// -------------------------------------------------
// subphase timer & counter
      A     M    103.0;

// -------------------------------------------------
// subphase actuator
      A     M    103.3;

// -------------------------------------------------
// subphase transition
      CLR   ;
      =     M    103.1;
      JU    COMM;
NETWORK
TITLE =phase 32: CIP Push Out
//SFM   Use                                 Datatype        UoM
//----+-------------------------------------------------------------------------
// 00 : Watch Dog Time                      Duration        min
// 01 : Step Time                           Duration        min
// 06 : Delay Switchpoint                   Duration        s
// 15 : Amount                              Value           m3
// 26 : CIP Step On Condition               Enumeration     min
// 27 : CIP Prerun                          Enumeration     min
// 28 : CIP Return                          Enumeration     min
// 29 : CIP Pump Speed                      Value           %
// 30 : CIP Return Temperature              Value           °C
// 32 : CIP Return Conductivity             Value           mS
// 34 : CIP Prerun Flow                     Value           m3/h
// 35 : CIP Prerun Pressure                 Value           bar
// 37 : CIP Pump Mode                       Enumeration     min
X32:  SET   ;
// ---------------------------------------------------------------------------
// General CM evaluation
      CALL FC   150 (
           ChkType                  := 3,
           ChkOK                    := #ChkOK);

      AN    #ChkOK;
      S     M    120.3;

// ---------------------------------------------------------------------------
// index evaluation: CIP Step On Condition
      CALL FC    45 (
           SFM                      := #U.Seq.SFM[26].Sp,
           Indexes                  := #S2I.SFM26);

// ---------------------------------------------------------------------------
// index evaluation: CIP Prerun
      CALL FC    45 (
           SFM                      := #U.Seq.SFM[27].Sp,
           Indexes                  := #S2I.SFM27);

// ---------------------------------------------------------------------------
// index evaluation: CIP Return
      CALL FC    45 (
           SFM                      := #U.Seq.SFM[28].Sp,
           Indexes                  := #S2I.SFM28);

// ---------------------------------------------------------------------------
// index evaluation: CIP Pump Mode
      CALL FC    45 (
           SFM                      := #U.Seq.SFM[37].Sp,
           Indexes                  := #S2I.SFM37);

// ---------------------------------------------------------------------------
// general functions
      AN    M    121.2;
      A     M    102.3;
      =     #RRel;

// ---------------------------------------------------------------------------
// messages
// ---------------------------------------------------------------------------
// timer & counter
      A     M    102.0;

// ---------------------------------------------------------------------------
// pause timer
      ON    M    102.3;
      O     M    150.0;
      S     M    140.0; // Step Time

      ON    M    102.3;
      O     M    150.5;
      S     M    140.5; // Delay Switchpoint

// ---------------------------------------------------------------------------
// communication

// ---------------------------------------------------------------------------
// control modules
      A     M    102.3;

// ---------------------------------------------------------------------------
// transition condition
      A     #SubStepMaxD;
      =     M    102.1;

// subphase evaluation
      L     MW   110;
      JL    D200;
      JU    COMM; // subphase  0:
// ---------------------------------------------------------------------------
D200: SET   ;
      S     M    110.7; // Error unknown subphase
      JU    COMM;
NETWORK
TITLE =phase 34: CIP Rinsing
//SFM   Use                                 Datatype        UoM
//----+-------------------------------------------------------------------------
// 00 : Watch Dog Time                      Duration        min
// 01 : Step Time                           Duration        min
// 05 : Substep Time                        Duration        s
// 06 : Delay Switchpoint                   Duration        s
// 15 : Amount                              Value           m3
// 27 : CIP Prerun                          Enumeration     min
// 28 : CIP Return                          Enumeration     min
// 29 : CIP Pump Speed                      Value           %
// 30 : CIP Return Temperature              Value           °C
// 32 : CIP Return Conductivity             Value           mS
// 34 : CIP Prerun Flow                     Value           m3/h
// 35 : CIP Prerun Pressure                 Value           bar
// 37 : CIP Pump Mode                       Enumeration     min
// 59 : Interval Counter                    Value           No.
X34:  SET   ;
// ---------------------------------------------------------------------------
// General CM evaluation
      CALL FC   150 (
           ChkType                  := 3,
           ChkOK                    := #ChkOK);

      AN    #ChkOK;
      S     M    120.3;

// ---------------------------------------------------------------------------
// index evaluation: CIP Prerun
      CALL FC    45 (
           SFM                      := #U.Seq.SFM[27].Sp,
           Indexes                  := #S2I.SFM27);

// ---------------------------------------------------------------------------
// index evaluation: CIP Return
      CALL FC    45 (
           SFM                      := #U.Seq.SFM[28].Sp,
           Indexes                  := #S2I.SFM28);

// ---------------------------------------------------------------------------
// index evaluation: CIP Pump Mode
      CALL FC    45 (
           SFM                      := #U.Seq.SFM[37].Sp,
           Indexes                  := #S2I.SFM37);

// ---------------------------------------------------------------------------
// general functions
      AN    M    121.2;
      A     M    102.3;
      =     #RRel;

// ---------------------------------------------------------------------------
// messages
// ---------------------------------------------------------------------------
// timer & counter
      A     M    102.0;

// ---------------------------------------------------------------------------
// pause timer
      ON    M    102.3;
      O     M    150.0;
      S     M    140.0; // Step Time

      ON    M    102.3;
      O     M    150.4;
      S     M    140.4; // Substep Time

      ON    M    102.3;
      O     M    150.5;
      S     M    140.5; // Delay Switchpoint

// ---------------------------------------------------------------------------
// communication

// ---------------------------------------------------------------------------
// control modules
      A     M    102.3;

// ---------------------------------------------------------------------------
// transition condition
      A     #SubStepMaxD;
      =     M    102.1;

// ---------------------------------------------------------------------------
// ---------------------------------------------------------------------------
// subphase repeat function
//      A     #SubStepMax
//      JCN  Y34
//      L     1
//      T     "SOSubStepNew"
//Y34:  SET

// subphase evaluation
      L     MW   110;
      JL    D400;
      JU    COMM; // subphase  0:
      JU    D401; // subphase  1: Pause
      JU    D402; // subphase  2: Main
      JU    D403; // subphase  3: Expulse
      JU    D404; // subphase  4: Seat Lift
      JU    D400; // subphase  5:
      JU    D406; // subphase  6: Shaft Rinse
      JU    D407; // subphase  7: Drain
// ---------------------------------------------------------------------------
D400: SET   ;
      S     M    110.7; // Error unknown subphase
      JU    COMM;

// subphase 1: Pause
D401: SET   ;

// -------------------------------------------------
// subphase timer & counter
      A     M    103.0;

// -------------------------------------------------
// subphase actuator
      A     M    103.3;

// -------------------------------------------------
// subphase transition
      CLR   ;
      =     M    103.1;
      JU    COMM;

// subphase 2: Main
D402: SET   ;

// -------------------------------------------------
// subphase timer & counter
      A     M    103.0;

// -------------------------------------------------
// subphase actuator
      A     M    103.3;

// -------------------------------------------------
// subphase transition
      CLR   ;
      =     M    103.1;
      JU    COMM;

// subphase 3: Expulse
D403: SET   ;

// -------------------------------------------------
// subphase timer & counter
      A     M    103.0;

// -------------------------------------------------
// subphase actuator
      A     M    103.3;

// -------------------------------------------------
// subphase transition
      CLR   ;
      =     M    103.1;
      JU    COMM;

// subphase 4: Seat Lift
D404: SET   ;

// -------------------------------------------------
// subphase timer & counter
      A     M    103.0;

// -------------------------------------------------
// subphase actuator
      A     M    103.3;

// -------------------------------------------------
// subphase transition
      CLR   ;
      =     M    103.1;
      JU    COMM;

// subphase 6: Shaft Rinse
D406: SET   ;

// -------------------------------------------------
// subphase timer & counter
      A     M    103.0;

// -------------------------------------------------
// subphase actuator
      A     M    103.3;

// -------------------------------------------------
// subphase transition
      CLR   ;
      =     M    103.1;
      JU    COMM;

// subphase 7: Drain
D407: SET   ;

// -------------------------------------------------
// subphase timer & counter
      A     M    103.0;

// -------------------------------------------------
// subphase actuator
      A     M    103.3;

// -------------------------------------------------
// subphase transition
      CLR   ;
      =     M    103.1;
      JU    COMM;
NETWORK
TITLE =phase 36: CIP Drain
//SFM   Use                                 Datatype        UoM
//----+-------------------------------------------------------------------------
// 00 : Watch Dog Time                      Duration        Min
// 04 : Delay Empty                         Duration        #sec
X36:  SET   ;
// ---------------------------------------------------------------------------
// General CM evaluation
      CALL FC   150 (
           ChkType                  := 3,
           ChkOK                    := #ChkOK);

      AN    #ChkOK;
      S     M    120.3;

// ---------------------------------------------------------------------------
// general functions
      AN    M    121.2;
      A     M    102.3;
      =     #RRel;

// ---------------------------------------------------------------------------
// messages
// ---------------------------------------------------------------------------
// timer & counter
      A     M    102.0;

// ---------------------------------------------------------------------------
// pause timer
      ON    M    102.3;
      O     M    150.3;
      S     M    140.3; // Delay Empty

// ---------------------------------------------------------------------------
// communication

// ---------------------------------------------------------------------------
// control modules
      A     M    102.3;

// ---------------------------------------------------------------------------
// transition condition
      A     #SubStepMaxD;
      =     M    102.1;

// subphase evaluation
      L     MW   110;
      JL    D600;
      JU    COMM; // subphase  0:
// ---------------------------------------------------------------------------
D600: SET   ;
      S     M    110.7; // Error unknown subphase
      JU    COMM;
NETWORK
TITLE =phase 40: CIP End
//SFM   Use                                 Datatype        UoM
//----+-------------------------------------------------------------------------
// 00 : Watch Dog Time                      Duration        min
X40:  SET   ;
// ---------------------------------------------------------------------------
// General CM evaluation
      CALL FC   150 (
           ChkType                  := 3,
           ChkOK                    := #ChkOK);

      AN    #ChkOK;
      S     M    120.3;

// ---------------------------------------------------------------------------
// general functions
      AN    M    121.2;
      A     M    102.3;
      =     #RRel;

// ---------------------------------------------------------------------------
// messages
// ---------------------------------------------------------------------------
// timer & counter
      A     M    102.0;

// ---------------------------------------------------------------------------
// pause timer
// ---------------------------------------------------------------------------
// communication

// ---------------------------------------------------------------------------
// control modules
      A     M    102.3;

// ---------------------------------------------------------------------------
// transition condition
      A     #SubStepMaxD;
      =     M    102.1;

// subphase evaluation
      L     MW   110;
      JL    E000;
      JU    COMM; // subphase  0:
// ---------------------------------------------------------------------------
E000: SET   ;
      S     M    110.7; // Error unknown subphase
      JU    COMM;

NETWORK
TITLE =End Of Sequence Organisation

COMM: SET   ;

// ---------------------------------------------------------------------------
// pause timer unit parameter

// Request Mole Water
      O     DB250.DBX  182.6;
      S     DB155.DBX   27.2;

      AN    DB1595.DBX   26.4; // Molchwasser
      R     DB250.DBX  188.0;

// Quelle
      L     DB155.DBW  254;
      L     1000;
      *I    ;
      T     #iTmp;

      L     0;
      T     #U.Seq.SFM[14].Sp;
      L     DB155.DBW  256;
      <I    ;
      JCN   ntru;
      L     #iTmp;
      +I    ;
      ITD   ;
      DTR   ;
      T     #U.Seq.SFM[14].Sp;
ntru: NOP   0;


NETWORK
TITLE =General Post Phase Controls
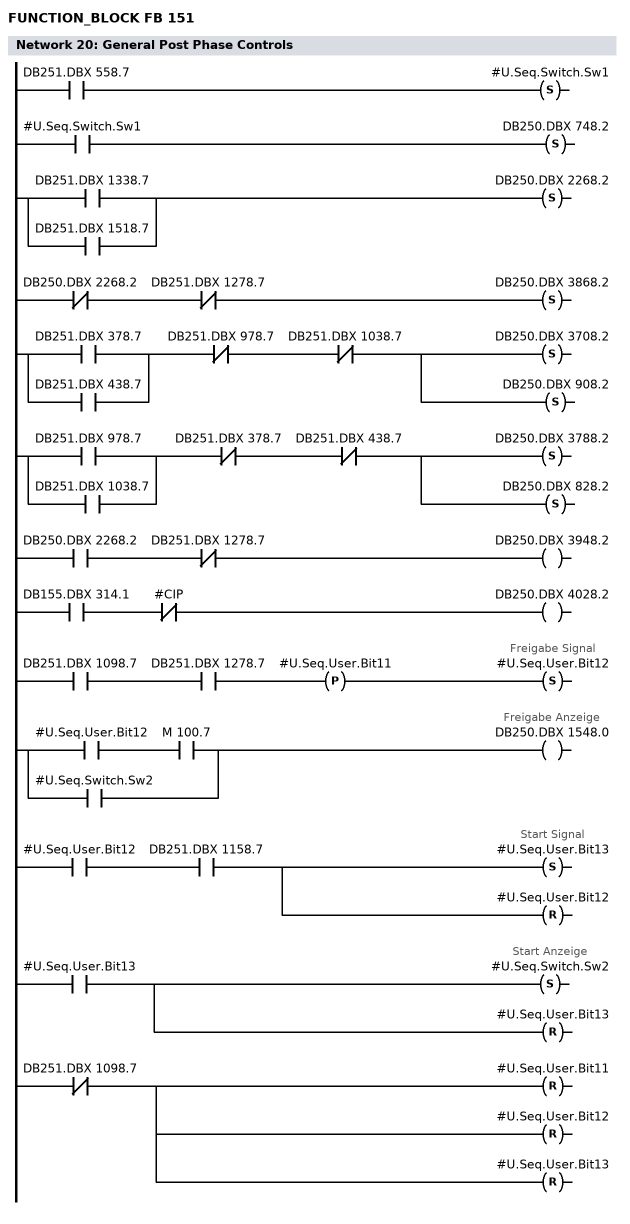

      NOP   0;

// ---------------------------------------------------------------------------
// general postphase controls
// Molchsignale  SR
      A     DB251.DBX  558.7;
      S     #U.Seq.Switch.Sw1;

      A     #U.Seq.Switch.Sw1;
      S     DB250.DBX  748.2;

// Molch Schwenkbogen auf CIP
      A     DB251.DBX 1338.7;
      O     DB251.DBX 1518.7;
      S     DB250.DBX 2268.2;

//Molch Bereit für Produktion
      AN    DB250.DBX 2268.2;
      AN    DB251.DBX 1278.7;
      S     DB250.DBX 3868.2;

//Molch im Sirupraum
      O     DB251.DBX  378.7;
      O     DB251.DBX  438.7;
      AN    DB251.DBX  978.7;
      AN    DB251.DBX 1038.7;
      S     DB250.DBX 3708.2;
      S     DB250.DBX  908.2;

//Molch an der Anlage
      O     DB251.DBX  978.7;
      O     DB251.DBX 1038.7;
      AN    DB251.DBX  378.7;
      AN    DB251.DBX  438.7;
      S     DB250.DBX 3788.2;
      S     DB250.DBX  828.2;

// Molch bereit für CIP
      A     DB250.DBX 2268.2;
      AN    DB251.DBX 1278.7;
      =     DB250.DBX 3948.2;

// Sirupanforderung
      A     DB155.DBX  314.1;
      AN    #CIP;
      =     DB250.DBX 4028.2;

// Molchsignale  A
      A     DB251.DBX 1098.7;
      A     DB251.DBX 1278.7;
      FP    #U.Seq.User.Bit11;
      S     #U.Seq.User.Bit12; // Freigabe Signal

      A     #U.Seq.User.Bit12;
      A     M    100.7;
      O     #U.Seq.Switch.Sw2;
      =     DB250.DBX 1548.0; // Freigabe Anzeige

      A     #U.Seq.User.Bit12;
      A     DB251.DBX 1158.7;
      S     #U.Seq.User.Bit13; // Start Signal
      R     #U.Seq.User.Bit12;

      A     #U.Seq.User.Bit13;
      S     #U.Seq.Switch.Sw2; // Start Anzeige
      R     #U.Seq.User.Bit13;

      AN    DB251.DBX 1098.7;
      R     #U.Seq.User.Bit11;
      R     #U.Seq.User.Bit12;
      R     #U.Seq.User.Bit13;



NETWORK
TITLE =Process Status Management

      NOP   0;
// ---------------------------------------------------------------------------
// Signal Control

      OPN   DB   500;
      L     #UnitNo;
      L     32; //U Structure Length
      *I    ;
      L     20; //DB Heading Offset
      +I    ;
      SLD   3;
      LAR2  ;

// -------------------------------------------------
// Maintenance
      A     #U.Seq.Switch.Sw31;
      OPN   DB   500;
      =     DBX [AR2,P#0.0]; //"PStatD".U[#UnitNo].MTNC
// -------------------------------------------------
// CIP Required
// -------------------------------------------------
// CIP Active
// -------------------------------------------------
// CIP Clean
// -------------------------------------------------
// SIP Required
// -------------------------------------------------
// SIP Active
// -------------------------------------------------
// SIP Clean
// -------------------------------------------------
// Full
      A     DB155.DBX   26.2;
      OPN   DB   500;
      =     DBX [AR2,P#0.7]; //"PStatD".U[#UnitNo].FULL
// -------------------------------------------------
// Filling
      A     DB155.DBX   26.1;
      OPN   DB   500;
      =     DBX [AR2,P#1.0]; //"PStatD".U[#UnitNo].FILL
// -------------------------------------------------
// Ready For Filling
      A     DB155.DBX   26.0;
      OPN   DB   500;
      =     DBX [AR2,P#1.1]; //"PStatD".U[#UnitNo].RFFI
// -------------------------------------------------
// Empty
      A     DB155.DBX   26.5;
      OPN   DB   500;
      =     DBX [AR2,P#1.2]; //"PStatD".U[#UnitNo].EMTY
// -------------------------------------------------
// Emptying
      A     DB155.DBX   26.4;
      OPN   DB   500;
      =     DBX [AR2,P#1.3]; //"PStatD".U[#UnitNo].EMTI
// -------------------------------------------------
// Ready For Emptying
      A     DB155.DBX   26.3;
      OPN   DB   500;
      =     DBX [AR2,P#1.4]; //"PStatD".U[#UnitNo].RFEM
// -------------------------------------------------
// Reserved
//      A     #ComXYZ
//      OPN   "PStatD"
//      =     DBX [AR2,P#1.5]             //"PStatD".U[#UnitNo].RESV
// -------------------------------------------------
// Production
// -------------------------------------------------
// Used

// -------------------------------------------------
// PStat Function Call

      CALL FC   500 (
           UnitNo                   := #UnitNo,
           PStatModVal              := DB255.DBD  234);

NETWORK
TITLE =Unit Hold Request and Messages

      SET   ;

// ---------------------------------------------------------------------------
// Set unit to "hold" if maintenance
      AN    #U.Seq.Switch.Sw31; // maintenance !
      JC    NCO1;
      S     M    120.3;
      L     998; // "Unit in maintenance !"
      T     MD    90;

// ---------------------------------------------------------------------------
// Set unit to "hold" if emergency stop
NCO1: A     #EStopOK;
      JC    NCO2;
      S     M    120.3;
      L     999; // "Emergency stop !"
      T     MD    90;
NCO2: NOP   0;

END_FUNCTION_BLOCK

FUNCTION_BLOCK FB 153
TITLE =C05: Syrup Transfer x
AUTHOR : Woermann
FAMILY : BOTEC_F1
NAME : C05E
VERSION : 1.2
CODE_VERSION1


VAR
  U : UDT 151;
END_VAR
VAR_TEMP
  CIP : BOOL ;	//CIP active
  UNIM : BOOL ;	//Unit Not In Maintenance
  GenRel : BOOL ;	//general OK (emergency and maintenance OK)
  EStopOK : BOOL ;	//emergency OK
  UnitNo : INT ;	//unit number
  xTmp : BOOL ;	//Temporary Bool
  iTmp : INT ;	//Temporary INT
  rTmp : REAL ;	//Temporary REAL
  dTmp : DINT ;	//Temporary DINT (free for general use)
  RetValInt : INT ;	//return value
  ComCIP1 : BOOL ;	//CIP1 in use
  ComCIP3 : BOOL ;	//CIP3 in use
END_VAR
BEGIN
NETWORK
TITLE =General


      SET   ;
// Simulation ---------------------------------------------------------------
      A     #U.Seq.User.Bit63;
      CC    FB   159; // "C05Sim"
      A     #U.Seq.Sim;
      =     #U.Seq.User.Bit63; //Help bit for simulation

// get unit number ----------------------------------------------------------
      L     DB150.DBW    0;
      L     DB155.DBW   16;
      T     #UnitNo;

// CIP ----------------------------------------------------------------------
      L     #U.Seq.ProgNo;
      L     0;
      <D    ;
      =     #CIP;

// emergency OK -------------------------------------------------------------
      A     DB155.DBX   27.0; //Emergency Stop OK
      =     #EStopOK;

// Write Unit in Maintenance ------------------------------------------------

      AN    #U.Seq.Switch.Sw31;
      =     #UNIM;

// emergency and maintenance OK ---------------------------------------------
      A     #EStopOK;
      A     #UNIM;
      =     #GenRel;

// communication ------------------------------------------------------------
      UC    FB   155; // U103Com

NETWORK
TITLE =Universal Value

      NOP   0;

// ----------------------------------------------------------
// unv001 Process Status
// ----------------------------------------------------------
// process value to UnV
//      L     0.000000e+000
//      T     "C05UnVD".unv001.ValExt

// ----------------------------------------------------------
// unv002 Universal Value 02
// ----------------------------------------------------------
// process value to UnV
//      L     0.000000e+000
//      T     "C05UnVD".unv002.ValExt

// ----------------------------------------------------------
// unv003 Universal Value 03
// ----------------------------------------------------------
// process value to UnV
//      L     0.000000e+000
//      T     "C05UnVD".unv003.ValExt

// ----------------------------------------------------------
// unv004 Universal Value 04
// ----------------------------------------------------------
// process value to UnV
//      L     0.000000e+000
//      T     "C05UnVD".unv004.ValExt

NETWORK
TITLE =Special Input

      NOP   0;

// ----------------------------------------------------------
// GOA_SKEG_31_oben GOA_SKEG_31_oben
// ----------------------------------------------------------
      CLR   ;
      =     DB251.DBX  261.4;
      =     DB251.DBX  261.5;

// ----------------------------------------------------------
// GOA_SKEG_32_unten GOA_SKEG_32_unten
// ----------------------------------------------------------
      CLR   ;
      =     DB251.DBX  321.4;
      =     DB251.DBX  321.5;

// ----------------------------------------------------------
// GOA_SKEG_1 GOA_SKEG_1
// ----------------------------------------------------------
      CLR   ;
      =     DB251.DBX  381.4;
      =     DB251.DBX  381.5;

// ----------------------------------------------------------
// GOA_SKEG_2 GOA_SKEG_2
// ----------------------------------------------------------
      CLR   ;
      =     DB251.DBX  441.4;
      =     DB251.DBX  441.5;

// ----------------------------------------------------------
// SK_KEG_Molch_Abbruch_DT MOLCH KEG Drucktaste Abbruch Sirupraum
// ----------------------------------------------------------
      CLR   ;
      =     DB251.DBX  501.4;
      =     DB251.DBX  501.5;

// ----------------------------------------------------------
// SK_KEG_START_Molch_LDT MOLCH KEG L-Drucktaste Start Sirupraum
// ----------------------------------------------------------
      CLR   ;
      =     DB251.DBX  561.4;
      =     DB251.DBX  561.5;

// ----------------------------------------------------------
// KEG_SK1_Handklappe KEG_SK1_Handklappe
// ----------------------------------------------------------
      CLR   ;
      =     DB251.DBX  621.4;
      =     DB251.DBX  621.5;

// ----------------------------------------------------------
// GOA_EKEG_31_oben GOA_EKEG_31_oben
// ----------------------------------------------------------
      CLR   ;
      =     DB251.DBX  861.4;
      =     DB251.DBX  861.5;

// ----------------------------------------------------------
// GOA_EKEG_32_unten GOA_EKEG_32_unten
// ----------------------------------------------------------
      CLR   ;
      =     DB251.DBX  921.4;
      =     DB251.DBX  921.5;

// ----------------------------------------------------------
// GOA_EKEG_3 GOA_EKEG_3
// ----------------------------------------------------------
      CLR   ;
      =     DB251.DBX  981.4;
      =     DB251.DBX  981.5;

// ----------------------------------------------------------
// GOA_EKEG_4 GOA_EKEG_4
// ----------------------------------------------------------
      CLR   ;
      =     DB251.DBX 1041.4;
      =     DB251.DBX 1041.5;

// ----------------------------------------------------------
// KEG_Freigabe_Molch_SS KEG_Freigabe_Molch_SS
// ----------------------------------------------------------
      CLR   ;
      =     DB251.DBX 1101.4;
      =     DB251.DBX 1101.5;

// ----------------------------------------------------------
// KEG_Molch_Start_LDT_I KEG_Molch_Start_LDT
// ----------------------------------------------------------
      CLR   ;
      =     DB251.DBX 1161.4;
      =     DB251.DBX 1161.5;

// ----------------------------------------------------------
// KEG_Stop_Molch_DT KEG_Stop_Molch_DT
// ----------------------------------------------------------
      CLR   ;
      =     DB251.DBX 1221.4;
      =     DB251.DBX 1221.5;

// ----------------------------------------------------------
// GOA_EKEG_5 GOA Handklappe am Paneel KEG Anlage (CO2)
// ----------------------------------------------------------
      CLR   ;
      =     DB251.DBX 1281.4;
      =     DB251.DBX 1281.5;

// ----------------------------------------------------------
// GOA_KEG_RR1 KEG RR Sirup Kreis 1 Schwenkbogen
// ----------------------------------------------------------
      CLR   ;
      =     DB251.DBX 1341.4;
      =     DB251.DBX 1341.5;

// ----------------------------------------------------------
// KEG_MIXER_BOGEN_22_24 KEG Mixer/KZE Schwenkbogen
// ----------------------------------------------------------
      CLR   ;
      =     DB251.DBX 1401.4;
      =     DB251.DBX 1401.5;

// ----------------------------------------------------------
// GOA_KEG_RR3 KEG RR Sirup Kreis 3 Schwenkbogen
// ----------------------------------------------------------
      CLR   ;
      =     DB251.DBX 1521.4;
      =     DB251.DBX 1521.5;

NETWORK
TITLE =Messages

      NOP   0;

// ----------------------------------------------------------
// msg001 Message 01
// ----------------------------------------------------------
      SET   ;
      R     DB257.DBX   80.7;
      =     DB257.DBX   81.4;

      CLR   ;
      =     DB257.DBX   82.7;

// ----------------------------------------------------------
// msg002 Message 02
// ----------------------------------------------------------
      SET   ;
      R     DB257.DBX  140.7;
      =     DB257.DBX  141.4;

      CLR   ;
      =     DB257.DBX  142.7;

// ----------------------------------------------------------
// msg003 Message 03
// ----------------------------------------------------------
      SET   ;
      R     DB257.DBX  200.7;
      =     DB257.DBX  201.4;

      CLR   ;
      =     DB257.DBX  202.7;

NETWORK
TITLE =Sequence organisation


// SFM supply ----------------------------------------------------------------

// sequencer ----------------------------------------------------------------

NETWORK
TITLE =Auto / Manual

      SET   ;
      AN    M    122.2;
      JC    MODE;
      AN    M    120.1;

// assign actuator mode
      AN    M    120.1;
      =     DB250.DBX  185.4;
      =     DB250.DBX  265.4;
      =     DB250.DBX  345.4;
      =     DB250.DBX  425.4;
      =     DB250.DBX  505.4;
      =     DB250.DBX  585.4;
      =     DB250.DBX  665.4;
      =     DB250.DBX  745.4;
      =     DB250.DBX  825.4;
      =     DB250.DBX  905.4;
      =     DB250.DBX  985.4;
      =     DB250.DBX 1065.4;
      =     DB250.DBX 1145.4;
      =     DB250.DBX 1225.4;
      =     DB250.DBX 1305.4;
      =     DB250.DBX 1385.4;
      =     DB250.DBX 1545.4;
      =     DB250.DBX 1625.4;
      =     DB250.DBX 1705.4;
      =     DB250.DBX 2265.4;
      =     DB250.DBX 2425.4;
      =     DB250.DBX 2505.4;
      =     DB250.DBX 2585.4;
      =     DB250.DBX 3705.4;
      =     DB250.DBX 3785.4;
      =     DB250.DBX 3865.4;
      =     DB250.DBX 3945.4;
      =     DB250.DBX 4025.4;

MODE: SET   ;

NETWORK
TITLE =KEG_MWV1 Ansteuerung KEG_MWV1
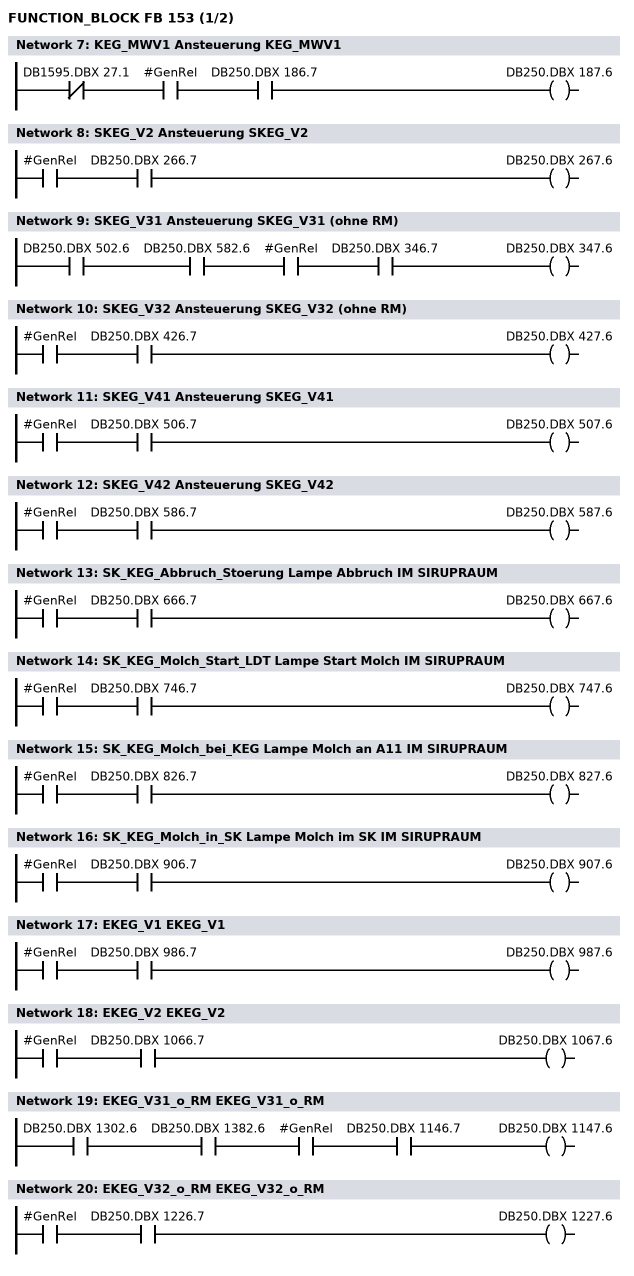

      AN    DB1595.DBX   27.1;
      A     #GenRel;
      A     DB250.DBX  186.7;
      =     DB250.DBX  187.6;

NETWORK
TITLE =SKEG_V2 Ansteuerung SKEG_V2

      A     #GenRel;
      A     DB250.DBX  266.7;
      =     DB250.DBX  267.6;
NETWORK
TITLE =SKEG_V31 Ansteuerung SKEG_V31 (ohne RM)

      A     DB250.DBX  502.6;
      A     DB250.DBX  582.6;

      A     #GenRel;
      A     DB250.DBX  346.7;
      =     DB250.DBX  347.6;

NETWORK
TITLE =SKEG_V32 Ansteuerung SKEG_V32 (ohne RM)

      A     #GenRel;
      A     DB250.DBX  426.7;
      =     DB250.DBX  427.6;
NETWORK
TITLE =SKEG_V41 Ansteuerung SKEG_V41

      A     #GenRel;
      A     DB250.DBX  506.7;
      =     DB250.DBX  507.6;
NETWORK
TITLE =SKEG_V42 Ansteuerung SKEG_V42

      A     #GenRel;
      A     DB250.DBX  586.7;
      =     DB250.DBX  587.6;
NETWORK
TITLE =SK_KEG_Abbruch_Stoerung Lampe Abbruch IM SIRUPRAUM

      A     #GenRel;
      A     DB250.DBX  666.7;
      =     DB250.DBX  667.6;
NETWORK
TITLE =SK_KEG_Molch_Start_LDT Lampe Start Molch IM SIRUPRAUM

      A     #GenRel;
      A     DB250.DBX  746.7;
      =     DB250.DBX  747.6;
NETWORK
TITLE =SK_KEG_Molch_bei_KEG Lampe Molch an A11 IM SIRUPRAUM

      A     #GenRel;
      A     DB250.DBX  826.7;
      =     DB250.DBX  827.6;
NETWORK
TITLE =SK_KEG_Molch_in_SK Lampe Molch im SK IM SIRUPRAUM

      A     #GenRel;
      A     DB250.DBX  906.7;
      =     DB250.DBX  907.6;
NETWORK
TITLE =EKEG_V1 EKEG_V1

      A     #GenRel;
      A     DB250.DBX  986.7;
      =     DB250.DBX  987.6;
NETWORK
TITLE =EKEG_V2 EKEG_V2

      A     #GenRel;
      A     DB250.DBX 1066.7;
      =     DB250.DBX 1067.6;
NETWORK
TITLE =EKEG_V31_o_RM EKEG_V31_o_RM

      A     DB250.DBX 1302.6;
      A     DB250.DBX 1382.6;

      A     #GenRel;
      A     DB250.DBX 1146.7;
      =     DB250.DBX 1147.6;
NETWORK
TITLE =EKEG_V32_o_RM EKEG_V32_o_RM

      A     #GenRel;
      A     DB250.DBX 1226.7;
      =     DB250.DBX 1227.6;
NETWORK
TITLE =EKEG_V41 EKEG_V41
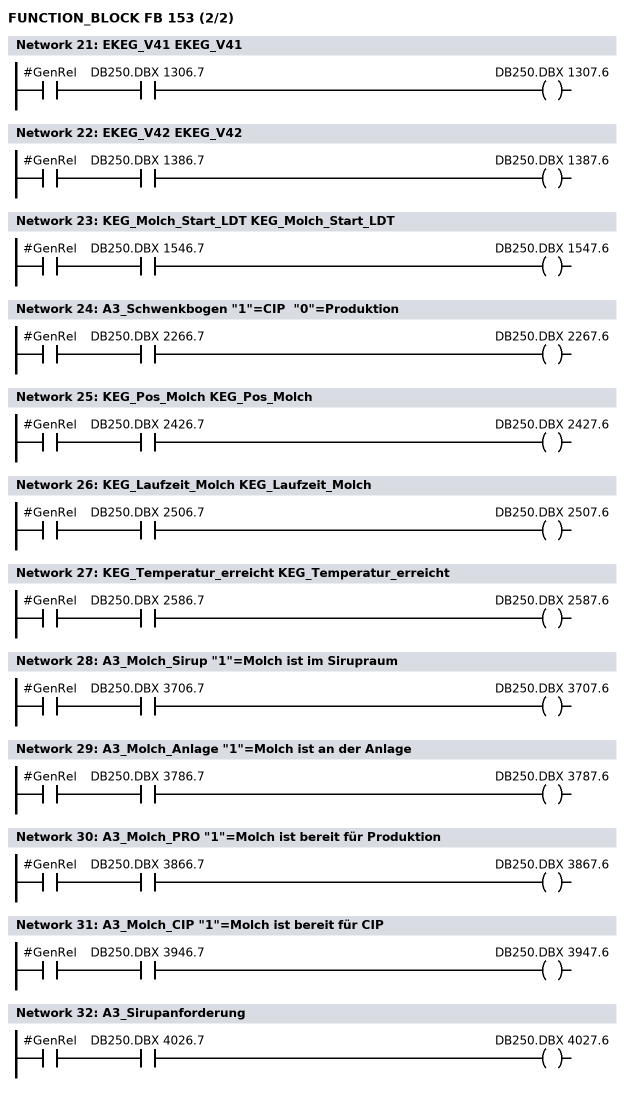

      A     #GenRel;
      A     DB250.DBX 1306.7;
      =     DB250.DBX 1307.6;
NETWORK
TITLE =EKEG_V42 EKEG_V42

      A     #GenRel;
      A     DB250.DBX 1386.7;
      =     DB250.DBX 1387.6;
NETWORK
TITLE =KEG_Molch_Start_LDT KEG_Molch_Start_LDT

      A     #GenRel;
      A     DB250.DBX 1546.7;
      =     DB250.DBX 1547.6;
NETWORK
TITLE =A3_Schwenkbogen "1"=CIP  "0"=Produktion

      A     #GenRel;
      A     DB250.DBX 2266.7;
      =     DB250.DBX 2267.6;
NETWORK
TITLE =KEG_Pos_Molch KEG_Pos_Molch

      A     #GenRel;
      A     DB250.DBX 2426.7;
      =     DB250.DBX 2427.6;
NETWORK
TITLE =KEG_Laufzeit_Molch KEG_Laufzeit_Molch

      A     #GenRel;
      A     DB250.DBX 2506.7;
      =     DB250.DBX 2507.6;
NETWORK
TITLE =KEG_Temperatur_erreicht KEG_Temperatur_erreicht

      A     #GenRel;
      A     DB250.DBX 2586.7;
      =     DB250.DBX 2587.6;
NETWORK
TITLE =A3_Molch_Sirup "1"=Molch ist im Sirupraum

      A     #GenRel;
      A     DB250.DBX 3706.7;
      =     DB250.DBX 3707.6;
NETWORK
TITLE =A3_Molch_Anlage "1"=Molch ist an der Anlage

      A     #GenRel;
      A     DB250.DBX 3786.7;
      =     DB250.DBX 3787.6;
NETWORK
TITLE =A3_Molch_PRO "1"=Molch ist bereit für Produktion

      A     #GenRel;
      A     DB250.DBX 3866.7;
      =     DB250.DBX 3867.6;
NETWORK
TITLE =A3_Molch_CIP "1"=Molch ist bereit für CIP

      A     #GenRel;
      A     DB250.DBX 3946.7;
      =     DB250.DBX 3947.6;
NETWORK
TITLE =A3_Sirupanforderung

      A     #GenRel;
      A     DB250.DBX 4026.7;
      =     DB250.DBX 4027.6;
END_FUNCTION_BLOCK

FUNCTION_BLOCK FB 155
TITLE =C05: Syrup Transfer x
AUTHOR : Woermann
FAMILY : BOTEC_F1
NAME : C05Comm
VERSION : 0.1
CODE_VERSION1


VAR
  U : UDT 151;
END_VAR
VAR_TEMP
  iRetVal : INT ;	//return value as integer
  wRetVal : WORD ;	//return value as word
  Run : BOOL ;	//Unit in "RUN" mode
  EStopOK : BOOL ;	//Emergency Stop OK
  CIP : BOOL ;	//CIP Program Selected
  ComCIP : BOOL ;	//Communication with CIP Active
  xTmp : BOOL ;	//Temporary BOOL (free for general use)
  iTmp : INT ;	//Temporary INT (free for general use)
  rTmp : REAL ;	//Temporary REAL (free for general use)
  dTmp : DINT ;	//Temporary DINT (free for general use)
  UnitNo : INT ;	//Unit Number
  EquipmentID : INT ;	//Equipment ID
  Prid : DINT ;	//Process ID
  SFM36 : STRUCT 	//CIP Pump Mode
   I00 : BOOL ;	// Off
   I01 : BOOL ;	// Flow
   I02 : BOOL ;	// Pressure
   I03 : BOOL ;	// Fix Speed
   I04 : BOOL ;
   I05 : BOOL ;
   I06 : BOOL ;
   I07 : BOOL ;
   I08 : BOOL ;
   I09 : BOOL ;
   I10 : BOOL ;
   I11 : BOOL ;
   I12 : BOOL ;
   I13 : BOOL ;
   I14 : BOOL ;
   I15 : BOOL ;
   I16 : BOOL ;
   I17 : BOOL ;
   I18 : BOOL ;
   I19 : BOOL ;
   I20 : BOOL ;
   I21 : BOOL ;
   I22 : BOOL ;
   I23 : BOOL ;
   I24 : BOOL ;
   I25 : BOOL ;
   I26 : BOOL ;
   I27 : BOOL ;
   I28 : BOOL ;
   I29 : BOOL ;
   I30 : BOOL ;
   I31 : BOOL ;
  END_STRUCT ;
  iPLC : INT ;
  iUnit : INT ;
  rUnitNo : REAL ;
  DSTUnit : INT ;	//Destination Unit
  SRCUnit : INT ;
  STBYUnit : INT ;
  rEquipmentID : REAL ;
END_VAR
BEGIN
NETWORK
TITLE =general

      SET   ;

// unit & equipment number ---------------------------------------------------
      L     DB150.DBW    0;
      L     DB155.DBW   16;
      T     #UnitNo;

      L     DB155.DBW   14;
      L     1000;
      *I    ;
      L     #UnitNo;
      +I    ;
      T     #EquipmentID;

// CIP ----------------------------------------------------------------------
      L     DB155.DBW   18;
      L     0;
      <I    ;
      =     #CIP;

// Communicating Units-------------------------------------------------------
      L     DB155.DBD   10;
      L     DB155.DBD  106;
      ==D   ;
      =     #ComCIP;

// ... General Unit ----------/

      CALL SFC   20 (
           SRCBLK                   := DB1995.Own,
           RET_VAL                  := #iRetVal,
           DSTBLK                   := DB155.GEN);

// emergency OK -------------------------------------------------------------
      A     DB155.DBX   75.0; //General Emergency Stop OK
      =     #EStopOK;

NETWORK
TITLE =read other unit's data

      SET   ;


//----------------------------------------
// Communication Packaging Plant
//----------------------------------------
      L     #U.Seq.Prop.Index0; // Source
      ITD   ;
      DTR   ;
      T     #rTmp;

      CALL FC   950 (
           EquipmentNo              := #rTmp,
           PLCNo                    := #iPLC,
           UnitNo                   := #iUnit);

      CALL FC   563 (
           ActReq                   := M    101.0,
           PLCNo                    := #iPLC,
           SourceUnitNo             := #iUnit,
           IsTUnit                  := FALSE,
           DstComDRec               := DB155.DST,
           RET_VAL                  := #wRetVal);


//----------------------------------------
// Communication Mixing Emptying
//----------------------------------------
      L     #U.Seq.SFM[14].Sp; // Source
      T     #rTmp;

      CALL FC   950 (
           EquipmentNo              := #rTmp,
           PLCNo                    := #iPLC,
           UnitNo                   := #iUnit);

// Select
      L     DB1995.DBD  250;
      L     DB155.DBD   10;
      ==D   ;
      AN    DB1995.DBX  264.7;
      JC    MTE1;
      L     DB1995.DBD  298;
      L     DB155.DBD   10;
      ==D   ;
      AN    DB1995.DBX  312.7;
      JC    MTE2;
      L     DB1995.DBD  346;
      L     DB155.DBD   10;
      ==D   ;
      AN    DB1995.DBX  360.7;
      JC    MTE3;
      L     DB1995.DBD  394;
      L     DB155.DBD   10;
      ==D   ;
      AN    DB1995.DBX  408.7;
      JC    MTE4;
      L     DB1995.DBD 1066;
      L     DB155.DBD   10;
      ==D   ;
      AN    DB1995.DBX 1080.7;
      JC    KZES;
      JU    ELS1;
// Case
MTE1: NOP   0;
      CALL SFC   20 (
           SRCBLK                   := DB1995.MTE1,
           RET_VAL                  := #iTmp,
           DSTBLK                   := DB155.SRC);
      JU    FIN1;
MTE2: NOP   0;
      CALL SFC   20 (
           SRCBLK                   := DB1995.MTE2,
           RET_VAL                  := #iTmp,
           DSTBLK                   := DB155.SRC);
      JU    FIN1;
MTE3: NOP   0;
      CALL SFC   20 (
           SRCBLK                   := DB1995.MTE3,
           RET_VAL                  := #iTmp,
           DSTBLK                   := DB155.SRC);
      JU    FIN1;
MTE4: NOP   0;
      CALL SFC   20 (
           SRCBLK                   := DB1995.MTE4,
           RET_VAL                  := #iTmp,
           DSTBLK                   := DB155.SRC);
      JU    FIN1;
KZES: NOP   0;
      CALL SFC   20 (
           SRCBLK                   := DB1995.P01U007,
           RET_VAL                  := #iTmp,
           DSTBLK                   := DB155.SRC);
      JU    FIN1;
ELS1: L     0;
      T     #rTmp;
      CALL SFC   21 (
           BVAL                     := #rTmp,
           RET_VAL                  := #iTmp,
           BLK                      := DB155.SRC);
FIN1: NOP   0;

// Anlage
// Select
      L     #UnitNo;
      L     103;
      ==I   ;
      JC    AN03;
      L     #UnitNo;
      L     105;
      ==I   ;
      JC    AN05;
      L     #UnitNo;
      L     107;
      ==I   ;
      JC    AN07;
      L     #UnitNo;
      L     109;
      ==I   ;
      JC    AN09;
      L     #UnitNo;
      L     112;
      ==I   ;
      JC    AN12;
      L     #UnitNo;
      L     114;
      ==I   ;
      JC    AN14;
      JU    ELS2;
// Case
AN03: NOP   0;
      CALL SFC   20 (
           SRCBLK                   := DB1995.P01U153,
           RET_VAL                  := #iTmp,
           DSTBLK                   := DB155.P01ANL);
      JU    FIN2;
AN05: NOP   0;
      CALL SFC   20 (
           SRCBLK                   := DB1995.P01U155,
           RET_VAL                  := #iTmp,
           DSTBLK                   := DB155.P01ANL);
      JU    FIN2;
AN07: NOP   0;
      CALL SFC   20 (
           SRCBLK                   := DB1995.P01U157,
           RET_VAL                  := #iTmp,
           DSTBLK                   := DB155.P01ANL);
      JU    FIN2;
AN09: NOP   0;
      CALL SFC   20 (
           SRCBLK                   := DB1995.P01U159,
           RET_VAL                  := #iTmp,
           DSTBLK                   := DB155.P01ANL);
      JU    FIN2;
AN12: NOP   0;
      CALL SFC   20 (
           SRCBLK                   := DB1995.P01U162,
           RET_VAL                  := #iTmp,
           DSTBLK                   := DB155.P01ANL);
      JU    FIN2;
AN14: NOP   0;
      CALL SFC   20 (
           SRCBLK                   := DB1995.P01U164,
           RET_VAL                  := #iTmp,
           DSTBLK                   := DB155.P01ANL);
      JU    FIN2;
ELS2: L     0;
      T     #rTmp;
      CALL SFC   21 (
           BVAL                     := #rTmp,
           RET_VAL                  := #iTmp,
           BLK                      := DB155.P01ANL);
FIN2: NOP   0;

NETWORK
TITLE =external releases

      SET   ;
      =     DB250.DBX  106.7;
      =     DB250.DBX  186.7;
      =     DB250.DBX  266.7;
      =     DB250.DBX  346.7;
      =     DB250.DBX  426.7;
      =     DB250.DBX  506.7;
      =     DB250.DBX  586.7;
      =     DB250.DBX  666.7;
      =     DB250.DBX  746.7;
      =     DB250.DBX  826.7;
      =     DB250.DBX  906.7;
      =     DB250.DBX  986.7;
      =     DB250.DBX 1066.7;
      =     DB250.DBX 1146.7;
      =     DB250.DBX 1226.7;
      =     DB250.DBX 1306.7;
      =     DB250.DBX 1386.7;
      =     DB250.DBX 1466.7;
      =     DB250.DBX 1546.7;
      =     DB250.DBX 1626.7;
      =     DB250.DBX 1706.7;
      =     DB250.DBX 1786.7;
      =     DB250.DBX 1866.7;
      =     DB250.DBX 1946.7;
      =     DB250.DBX 2026.7;
      =     DB250.DBX 2106.7;
      =     DB250.DBX 2186.7;
      =     DB250.DBX 2266.7;
      =     DB250.DBX 2346.7;
      =     DB250.DBX 2426.7;
      =     DB250.DBX 2506.7;
      =     DB250.DBX 2586.7;
      =     DB250.DBX 2666.7;
      =     DB250.DBX 2746.7;
      =     DB250.DBX 2826.7;
      =     DB250.DBX 2906.7;
      =     DB250.DBX 2986.7;
      =     DB250.DBX 3066.7;
      =     DB250.DBX 3146.7;
      =     DB250.DBX 3226.7;
      =     DB250.DBX 3306.7;
      =     DB250.DBX 3386.7;
      =     DB250.DBX 3466.7;
      =     DB250.DBX 3546.7;
      =     DB250.DBX 3626.7;
      =     DB250.DBX 3706.7;
      =     DB250.DBX 3786.7;
      =     DB250.DBX 3866.7;
      =     DB250.DBX 3946.7;
      =     DB250.DBX 4026.7;

NETWORK
TITLE =write own unit data

      SET   ;

//-- CIP Communication ---------------------------------------
      AN    #U.Seq.Step0;
      AN    #U.Seq.PO.B30; // CIP Active (Slave)
      A     #ComCIP;
      JCN   NCIP;
//Conductivity CIP Return
      L     DB155.DBD  150;
      T     #U.Seq.SFM[32].Val;

//Temperature CIP Return
      L     DB155.DBD  146;
      T     #U.Seq.SFM[30].Val;

//CIP Prerun Pump SP

      CALL FC    45 (
           SFM                      := #U.Seq.SFM[36].Sp,
           Indexes                  := #SFM36);


      L     0.000000e+000;
      A     #SFM36.I01;
      =     DB155.DBX  171.7;
      JCN   pfc;
      L     #U.Seq.SFM[34].Sp;
pfc:  NOP   0;
      A     #SFM36.I02;
      =     DB155.DBX  172.0;
      JCN   ppc;
      L     #U.Seq.SFM[35].Sp;
ppc:  NOP   0;
      A     #SFM36.I03;
      =     DB155.DBX  171.6;
      JCN   pxc;
      L     #U.Seq.SFM[29].Sp;
pxc:  NOP   0;
      T     DB155.DBD  182;

//CIP Return
      L     #U.Seq.SFM[28].Sp;
      T     DB155.DBD  186;
      L     DB155.DBD  138;
      T     #U.Seq.SFM[28].Val;

//CIP Prerun
      L     #U.Seq.SFM[27].Sp;
      T     DB155.DBD  190;
      L     DB155.DBD  142;
      T     #U.Seq.SFM[27].Val;

// Write Own Data to CIP
      L     DB155.DBD   10;
      T     DB155.DBD  154;

      L     DB155.DBW   14;
      T     DB155.DBW  158;

      L     DB155.DBW   16;
      T     DB155.DBW  160;

      L     DB155.DBW   18;
      T     DB155.DBW  162;

      L     DB155.DBW   20;
      T     DB155.DBW  164;

      L     DB155.DBW   22;
      T     DB155.DBW  166;

      A     DB155.DBX   24.0;
      =     DB155.DBX  168.0;

      A     DB155.DBX   24.1;
      =     DB155.DBX  168.1;

      A     DB155.DBX   24.2;
      =     DB155.DBX  168.2;

      A     DB155.DBX   24.3;
      =     DB155.DBX  168.3;

      A     DB155.DBX   24.4;
      =     DB155.DBX  168.4;

      A     DB155.DBX   24.5;
      =     DB155.DBX  168.5;

      A     DB155.DBX   24.6;
      =     DB155.DBX  168.6;

      A     DB155.DBX   24.7;
      =     DB155.DBX  168.7;

// Copy Data to CIP
      CALL SFC   20 (
           SRCBLK                   := DB155.ToCIP,
           RET_VAL                  := #iRetVal,
           DSTBLK                   := DB155.ToCIP);

NCIP: NOP   0;

//Empty Signal
//A     "C05SpID".SpI.Sig //!!!! Insert correct Empty Signal !!!
      CLR   ;
      =     DB155.DBX   26.5;

//Full Signal
//A     "C05SpID".SpI.Sig //!!!! Insert correct Full Signal !!!
      CLR   ;
      =     DB155.DBX   26.2;

//CIP Program Selected
      A     #CIP;
      =     DB155.DBX   27.1;

// Emergency Stop
      A     #EStopOK; //If needed add or replace with own SpI
      =     DB155.DBX   27.0; //Emergency Stop OK


NETWORK
TITLE = read from other unit data



END_FUNCTION_BLOCK

FUNCTION_BLOCK FB 159
TITLE =C05: Syrup Transfer x
AUTHOR : Woermann
FAMILY : BOTEC_F1
NAME : C05Sim
VERSION : 0.1
CODE_VERSION1


VAR
  U : UDT 151;
END_VAR
VAR_TEMP
  CIP : BOOL ;	//CIP active
  xTmp : BOOL ;	//Temporary BOOL (free for general use)
  iTmp : INT ;	//Temporary INT (free for general use)
  rTmp : REAL ;	//Temporary REAL (free for general use)
  UnitNo : INT ;	//Unit Number
END_VAR
BEGIN
NETWORK
TITLE =General

      SET   ;
// get unit number ----------------------------------------------------------
      L     #U.Seq.UnitNo;
      T     #UnitNo;

// CIP ----------------------------------------------------------------------
      L     #U.Seq.ProgNo;
      L     0;
      <D    ;
      =     #CIP;

NETWORK
TITLE =Actuator

      A     #U.Seq.Sim;
      =     DB250.DBX  105.3;
      =     DB250.DBX  185.3;
      =     DB250.DBX  265.3;
      =     DB250.DBX  345.3;
      =     DB250.DBX  425.3;
      =     DB250.DBX  505.3;
      =     DB250.DBX  585.3;
      =     DB250.DBX  665.3;
      =     DB250.DBX  745.3;
      =     DB250.DBX  825.3;
      =     DB250.DBX  905.3;
      =     DB250.DBX  985.3;
      =     DB250.DBX 1065.3;
      =     DB250.DBX 1145.3;
      =     DB250.DBX 1225.3;
      =     DB250.DBX 1305.3;
      =     DB250.DBX 1385.3;
      =     DB250.DBX 1465.3;
      =     DB250.DBX 1545.3;
      =     DB250.DBX 1625.3;
      =     DB250.DBX 1705.3;
      =     DB250.DBX 1785.3;
      =     DB250.DBX 1865.3;
      =     DB250.DBX 1945.3;
      =     DB250.DBX 2025.3;
      =     DB250.DBX 2105.3;
      =     DB250.DBX 2185.3;
      =     DB250.DBX 2265.3;
      =     DB250.DBX 2345.3;
      =     DB250.DBX 2425.3;
      =     DB250.DBX 2505.3;
      =     DB250.DBX 2585.3;
      =     DB250.DBX 2665.3;
      =     DB250.DBX 2745.3;
      =     DB250.DBX 2825.3;
      =     DB250.DBX 2905.3;
      =     DB250.DBX 2985.3;
      =     DB250.DBX 3065.3;
      =     DB250.DBX 3145.3;
      =     DB250.DBX 3225.3;
      =     DB250.DBX 3305.3;
      =     DB250.DBX 3385.3;
      =     DB250.DBX 3465.3;
      =     DB250.DBX 3545.3;
      =     DB250.DBX 3625.3;
      =     DB250.DBX 3705.3;
      =     DB250.DBX 3785.3;
      =     DB250.DBX 3865.3;
      =     DB250.DBX 3945.3;
      =     DB250.DBX 4025.3;

NETWORK
TITLE =Special Input

      A     #U.Seq.Sim;
      =     DB251.DBX   81.3;
      =     DB251.DBX  141.3;
      =     DB251.DBX  201.3;
      =     DB251.DBX  261.3;
      =     DB251.DBX  321.3;
      =     DB251.DBX  381.3;
      =     DB251.DBX  441.3;
      =     DB251.DBX  501.3;
      =     DB251.DBX  561.3;
      =     DB251.DBX  621.3;
      =     DB251.DBX  681.3;
      =     DB251.DBX  741.3;
      =     DB251.DBX  801.3;
      =     DB251.DBX  861.3;
      =     DB251.DBX  921.3;
      =     DB251.DBX  981.3;
      =     DB251.DBX 1041.3;
      =     DB251.DBX 1101.3;
      =     DB251.DBX 1161.3;
      =     DB251.DBX 1221.3;
      =     DB251.DBX 1281.3;
      =     DB251.DBX 1341.3;
      =     DB251.DBX 1401.3;
      =     DB251.DBX 1461.3;
      =     DB251.DBX 1521.3;


NETWORK
TITLE =Counter

      A     #U.Seq.Sim;
      A     M    101.0;
      CLR   ;
NETWORK
TITLE =Analog Input

      A     #U.Seq.Sim;

NETWORK
TITLE =Universal Value

      A     #U.Seq.Sim;


NETWORK
TITLE =PID

      A     #U.Seq.Sim;

NETWORK
TITLE =Message

      A     #U.Seq.Sim;


NETWORK
TITLE =VLT

      A     #U.Seq.Sim;

END_FUNCTION_BLOCK

FUNCTION_BLOCK FB 161
TITLE =C06: CIP Line x
// NW  1 : phase and index evaluation
// NW  2 : phase  1: start position
// NW  3 : phase  4: Filling
// NW  4 : phase  5: Storage
// NW  5 : phase  8: Emptying
// NW  6 : phase 20: Quality Check
// NW  7 : phase 21: Prepare Tank
// NW  8 : phase 23: Connect Tank
// NW  9 : phase 31: CIP Start
// NW 10 : phase 32: CIP Prerun
// NW 11 : phase 33: CIP Return
// NW 12 : phase 34: CIP Rinsing
// NW 13 : phase 35: CIP Emptying
// NW 14 : phase 36: CIP Drain
// NW 15 : phase 40: CIP End
// NW 16 : end of sequence
// NW 17 : unit hold request
//SFM   Use                                 Datatype        UoM
//----+-------------------------------------------------------------------------
// 09 : Process Time                        Duration        min
// 40 : Density                             Value           kg/l
// 42 : Material                            Value
AUTHOR : Woermann
NAME : C06Seq
VERSION : 0.1
CODE_VERSION1


VAR
  U : UDT 161;
END_VAR
VAR_TEMP
  CIP : BOOL ;	//CIP active
  ComCIP : BOOL ;	//Communication With CIP Active
  ComXYZ : BOOL ;	//Communication With Unit XYZ
  RRel : BOOL ;	//Run Release
  EStopOK : BOOL ;	//emergency OK
  StepMax : BOOL ;	//StepMax (last) active
  SubStepMax : BOOL ;	//SubStepMax (last) active
  SubStepMaxD : BOOL ;	//SubStepMax (last) done
  ChkOK : BOOL ;	//SubStepMax (last) done
  xTmp : BOOL ;	//Temporary BOOL (free for general use)
  iTmp : INT ;	//Temporary INT (free for general use)
  dTmp : DINT ;	//Temporary DINT (free for general use)
  rTmp : REAL ;	//Temporary REAL (free for general use)
  dUnitNo : DINT ;	//Unit Number
  UnitNo : INT ;	//Unit Number
  EquipmentID : INT ;	//Equipment ID
  S2I : STRUCT 	//SFM to indexes
   SFM25 : STRUCT 	//CIP Way
    I00 : BOOL ;
    I01 : BOOL ;	//Water Tanks
    I02 : BOOL ;	//Packaging Plants
    I03 : BOOL ;	//CIP 1 Distribution
    I04 : BOOL ;	//CIP 3 Distribution
    I05 : BOOL ;	//Charcoal Filter
    I06 : BOOL ;	//Packaging Plant 5
    I07 : BOOL ;	//Packaging Plant 14
    I08 : BOOL ;	//CIP 2 Common
    I09 : BOOL ;	//KEG Plant / Wells
    I10 : BOOL ;
    I11 : BOOL ;
    I12 : BOOL ;
    I13 : BOOL ;
    I14 : BOOL ;
    I15 : BOOL ;
    I16 : BOOL ;
    I17 : BOOL ;
    I18 : BOOL ;
    I19 : BOOL ;
    I20 : BOOL ;
    I21 : BOOL ;
    I22 : BOOL ;
    I23 : BOOL ;
    I24 : BOOL ;
    I25 : BOOL ;
    I26 : BOOL ;
    I27 : BOOL ;
    I28 : BOOL ;
    I29 : BOOL ;
    I30 : BOOL ;
    I31 : BOOL ;
   END_STRUCT ;
   SFM26 : STRUCT 	//Cip Step On Condition
    I00 : BOOL ;	//Please Select
    I01 : BOOL ;	//Conductivity High
    I02 : BOOL ;	//Conductivity Low
    I03 : BOOL ;	//Time
    I04 : BOOL ;	//Amount
    I05 : BOOL ;	//Temperature High
    I06 : BOOL ;	//Temperature Low
    I07 : BOOL ;
    I08 : BOOL ;
    I09 : BOOL ;
    I10 : BOOL ;
    I11 : BOOL ;
    I12 : BOOL ;
    I13 : BOOL ;
    I14 : BOOL ;
    I15 : BOOL ;
    I16 : BOOL ;
    I17 : BOOL ;
    I18 : BOOL ;
    I19 : BOOL ;
    I20 : BOOL ;
    I21 : BOOL ;
    I22 : BOOL ;
    I23 : BOOL ;
    I24 : BOOL ;
    I25 : BOOL ;
    I26 : BOOL ;
    I27 : BOOL ;
    I28 : BOOL ;
    I29 : BOOL ;
    I30 : BOOL ;
    I31 : BOOL ;
   END_STRUCT ;
   SFM27 : STRUCT 	//Cip Prerun
    I00 : BOOL ;	//None
    I01 : BOOL ;	//Recovered Water
    I02 : BOOL ;	//Caustic
    I03 : BOOL ;
    I04 : BOOL ;	//Acid
    I05 : BOOL ;
    I06 : BOOL ;
    I07 : BOOL ;
    I08 : BOOL ;
    I09 : BOOL ;
    I10 : BOOL ;
    I11 : BOOL ;
    I12 : BOOL ;	//Fresh Water
    I13 : BOOL ;	//Warm Water
    I14 : BOOL ;
    I15 : BOOL ;
    I16 : BOOL ;
    I17 : BOOL ;
    I18 : BOOL ;
    I19 : BOOL ;
    I20 : BOOL ;
    I21 : BOOL ;
    I22 : BOOL ;
    I23 : BOOL ;
    I24 : BOOL ;
    I25 : BOOL ;
    I26 : BOOL ;
    I27 : BOOL ;
    I28 : BOOL ;
    I29 : BOOL ;
    I30 : BOOL ;
    I31 : BOOL ;
   END_STRUCT ;
   SFM28 : STRUCT 	//Cip Return
    I00 : BOOL ;	//None
    I01 : BOOL ;	//Recovered Water
    I02 : BOOL ;	//Caustic
    I03 : BOOL ;
    I04 : BOOL ;	//Acid
    I05 : BOOL ;
    I06 : BOOL ;
    I07 : BOOL ;
    I08 : BOOL ;
    I09 : BOOL ;
    I10 : BOOL ;
    I11 : BOOL ;
    I12 : BOOL ;	//Fresh Water
    I13 : BOOL ;	//Warm Water
    I14 : BOOL ;
    I15 : BOOL ;	//Drain
    I16 : BOOL ;
    I17 : BOOL ;
    I18 : BOOL ;
    I19 : BOOL ;
    I20 : BOOL ;
    I21 : BOOL ;
    I22 : BOOL ;
    I23 : BOOL ;
    I24 : BOOL ;
    I25 : BOOL ;
    I26 : BOOL ;
    I27 : BOOL ;
    I28 : BOOL ;
    I29 : BOOL ;
    I30 : BOOL ;
    I31 : BOOL ;
   END_STRUCT ;
   SFM37 : STRUCT 	//Cip Pump Mode
    I00 : BOOL ;	//Off
    I01 : BOOL ;	//Flow
    I02 : BOOL ;	//Pressure
    I03 : BOOL ;	//Fix Speed
    I04 : BOOL ;
    I05 : BOOL ;
    I06 : BOOL ;
    I07 : BOOL ;
    I08 : BOOL ;
    I09 : BOOL ;
    I10 : BOOL ;
    I11 : BOOL ;
    I12 : BOOL ;
    I13 : BOOL ;
    I14 : BOOL ;
    I15 : BOOL ;
    I16 : BOOL ;
    I17 : BOOL ;
    I18 : BOOL ;
    I19 : BOOL ;
    I20 : BOOL ;
    I21 : BOOL ;
    I22 : BOOL ;
    I23 : BOOL ;
    I24 : BOOL ;
    I25 : BOOL ;
    I26 : BOOL ;
    I27 : BOOL ;
    I28 : BOOL ;
    I29 : BOOL ;
    I30 : BOOL ;
    I31 : BOOL ;
   END_STRUCT ;
   SFM31 : STRUCT 	//Cip Distribution Circuit No
    I00 : BOOL ;	//Please Select
    I01 : BOOL ;	//Auto Select
    I02 : BOOL ;
    I03 : BOOL ;
    I04 : BOOL ;
    I05 : BOOL ;
    I06 : BOOL ;
    I07 : BOOL ;
    I08 : BOOL ;
    I09 : BOOL ;
    I10 : BOOL ;
    I11 : BOOL ;
    I12 : BOOL ;
    I13 : BOOL ;
    I14 : BOOL ;
    I15 : BOOL ;
    I16 : BOOL ;
    I17 : BOOL ;
    I18 : BOOL ;
    I19 : BOOL ;
    I20 : BOOL ;
    I21 : BOOL ;
    I22 : BOOL ;
    I23 : BOOL ;
    I24 : BOOL ;
    I25 : BOOL ;
    I26 : BOOL ;
    I27 : BOOL ;
    I28 : BOOL ;
    I29 : BOOL ;
    I30 : BOOL ;
    I31 : BOOL ;
   END_STRUCT ;
   SFM39 : STRUCT 	//Q-Status
    I00 : BOOL ;	//Please select
    I01 : BOOL ;	//released
    I02 : BOOL ;
    I03 : BOOL ;
    I04 : BOOL ;
    I05 : BOOL ;
    I06 : BOOL ;	//Ignore
    I07 : BOOL ;
    I08 : BOOL ;
    I09 : BOOL ;	//locked
    I10 : BOOL ;
    I11 : BOOL ;
    I12 : BOOL ;
    I13 : BOOL ;
    I14 : BOOL ;
    I15 : BOOL ;
    I16 : BOOL ;
    I17 : BOOL ;
    I18 : BOOL ;
    I19 : BOOL ;
    I20 : BOOL ;
    I21 : BOOL ;
    I22 : BOOL ;
    I23 : BOOL ;
    I24 : BOOL ;
    I25 : BOOL ;
    I26 : BOOL ;
    I27 : BOOL ;
    I28 : BOOL ;
    I29 : BOOL ;
    I30 : BOOL ;
    I31 : BOOL ;
   END_STRUCT ;
  END_STRUCT ;
  ComDST : BOOL ;	//Communication Water Transfer to Packaging Plant
  ComCIPDist : BOOL ;	//Communication with CIP Distribution
  ReqInlet : BOOL ;	//Request Inlet
  RelOutlet : BOOL ;	//Release Outlet
  PStat : UDT 500;
  Empty : BOOL ;	//Tank Empty
  ReqCTopUp : BOOL ;	//Request Caustic Top Up
  ReqATopUp : BOOL ;	//Request Acid Top Up
END_VAR
BEGIN
NETWORK
TITLE =Phase and Index Evaluation

      CLR   ;
      =     #RRel;
// ---------------------------------------------------------------------------
// write max used SFM's (last SFM number + 1)
      L     37;
      T     #U.SFMQuant;

// ---------------------------------------------------------------------------
// unit & equipment number
      L     MB   112;
      T     #UnitNo;

      L     DB165.DBW   14;
      L     1000;
      *I    ;
      L     #UnitNo;
      +I    ;
      T     #EquipmentID;

// ---------------------------------------------------------------------------
// CIP active
      L     MW   114;
      L     0;
      <I    ;
      =     #CIP;

// ---------------------------------------------------------------------------
// communicating units
      L     MD   124;
      L     DB165.DBD  106;
      ==D   ;
      =     #ComCIP;

      L     MD   124;
//      L     "UxxxComD".Own.PrId //!!! Fill in Communicating Unit Number
      ==D   ;
      =     #ComXYZ; //!!! Fill in Shortname for Communicating Unit

// ---------------------------------------------------------------------------
// process timer start
      SET   ;
      =     M    131.0;

// ---------------------------------------------------------------------------
// emergency OK
      A     DB165.DBX   27.0;
      =     #EStopOK;

// define last (Sub)Step active
      L     #U.Seq.StepMax;
      L     MW   104;
      ==I   ;
      =     #StepMax;

      L     #U.Seq.SubStepMax;
      L     MW   118;
      ==I   ;
      =     #SubStepMax;

      A     #SubStepMax;
      A     #U.Seq.SPD;
      AN    M    103.2;
      =     #SubStepMaxD;

// ---------------------------------------------------------------------------
// phase evaluation
      L     MW   108;
      JL    X0;
      JU    X0; // phase  0:
      JU    X1; // phase  1: start position
      JU    X0; // phase  2:
      JU    X0; // phase  3:
      JU    X0; // phase  4:
      JU    X0; // phase  5
      JU    X0; // phase  6:
      JU    X0; // phase  7:
      JU    X0; // phase  8:
      JU    X0; // phase  9:
      JU    X0; // phase 10:
      JU    X0; // phase 11:
      JU    X0; // phase 12:
      JU    X0; // phase 13:
      JU    X0; // phase 14:
      JU    X0; // phase 15:
      JU    X0; // phase 16:
      JU    X0; // phase 17:
      JU    X0; // phase 18:
      JU    X0; // phase 19:
      JU    X0; // phase 20:
      JU    X0; // phase 21:
      JU    X0; // phase 22:
      JU    X0; // phase 23:
      JU    X0; // phase 24:
      JU    X0; // phase 25:
      JU    X0; // phase 26:
      JU    X0; // phase 27:
      JU    X0; // phase 28:
      JU    X0; // phase 29:
      JU    X0; // phase 30:
      JU    X31; // phase 31: CIP Active
X0:   SET   ;
      S     M    108.7; // Error unknown phase
      JU    COMM;
NETWORK
TITLE =phase 1: startposition

X1:   SET   ;

// ---------------------------------------------------------------------------
// general functions
// ---------------------------------------------------------------------------
// reset signals
      A     M    102.2;
      R     #U.Seq.Switch.Sw1;
      R     #U.Seq.Switch.Sw2;

      L     0.000000e+000;
      T     #U.Seq.User.Real11;
      T     #U.Seq.User.Real12;
      T     #U.Seq.User.Real13;

      AN    M    102.0;
      =     M    161.0; // Reset Process Timer

      CALL FC   709 (// Reset "Simulation" And "Ignore"
           UnitNo                   := #UnitNo,// Of All Control Modules
           Enable                   := M    102.2);// At First Cycle of Startposition (Idle)

// ---------------------------------------------------------------------------
// reset counter ------------------------------------------------------------
      AN    M    102.0;
      S     DB262.DBX  181.4;

// ---------------------------------------------------------------------------
// start check --------------------------------------------------------------
      A     #CIP;
      JC    M010;

      CALL FC   160 (
           ChkType                  := 1,// production
           ChkOK                    := M    122.0);
      JU    COMM;

M010: CALL FC   160 (
           ChkType                  := 2,// CIP
           ChkOK                    := M    122.0);
      JU    COMM;
NETWORK
TITLE =phase 31: CIP Active
//SFM   Use                                 Datatype        UoM
//----+-------------------------------------------------------------------------
// 00 : Watch Dog Time                      Duration        min
// 25 : CIP Way                             Enumeration
// 27 : Cip Prerun                          Enumeration
// 28 : Cip Return                          Enumeration
// 29 : Cip Pump Speed                      Value           %
// 30 : Cip Return Temperature              Value           °C
// 32 : Cip Return Conductivity             Value           mS
// 33 : Cip Return Pump Speed               Value           %
// 34 : Cip Prerun Flow                     Value           m3/h
// 35 : Cip Prerun Pressure                 Value           bar
X31:  SET   ;
// ---------------------------------------------------------------------------
// General CM evaluation
      CALL FC   160 (
           ChkType                  := 3,
           ChkOK                    := #ChkOK);

      AN    #ChkOK;
      S     M    120.3;

// ---------------------------------------------------------------------------
// index evaluation: CIP Way
      CALL FC    45 (
           SFM                      := #U.Seq.SFM[25].Sp,
           Indexes                  := #S2I.SFM25);

// ---------------------------------------------------------------------------
// index evaluation: CIP Prerun
      CALL FC    45 (
           SFM                      := #U.Seq.SFM[27].Sp,
           Indexes                  := #S2I.SFM27);

// ---------------------------------------------------------------------------
// index evaluation: CIP Return
      CALL FC    45 (
           SFM                      := #U.Seq.SFM[28].Sp,
           Indexes                  := #S2I.SFM28);

// ---------------------------------------------------------------------------
// general functions
      AN    M    121.2;
      A     M    102.3;
      =     #RRel;

// ---------------------------------------------------------------------------
// messages
// ---------------------------------------------------------------------------
// timer & counter
// ---------------------------------------------------------------------------
// pause timer
// ---------------------------------------------------------------------------
// communication
// CIP Active
      A     M    102.0;
      =     DB165.DBX   27.4;
// CIP Run Release
      A     #RRel;
      =     DB165.DBX   27.5;

// ---------------------------------------------------------------------------
// control modules
// ---------------------------------------------------------------------------
// CIP Return ---
// ---------------------------------------------------------------------------
      L     DB165.DBD  138;
      T     #U.Seq.SFM[28].Sp;

// Circulation
      A     #S2I.SFM28.I16;
      A     DB165.DBX  124.7;
      A     #RRel;
      =     DB260.DBX 2588.0;

// Caustic
      A     #S2I.SFM28.I02;
      A     DB165.DBX  124.7;
      A     #RRel;
      =     DB260.DBX  748.0;

// Acid
      A     #S2I.SFM28.I04;
      A     DB165.DBX  124.7;
      A     #RRel;
      =     DB260.DBX  828.0;

// Hot Water
      A     #S2I.SFM28.I13;
      A     DB165.DBX  124.7;
      A     #RRel;
      =     DB260.DBX  908.0;

// Drain
      AN    DB260.DBX  748.0;
      AN    DB260.DBX  828.0;
      A     #S2I.SFM28.I15;
      A     DB165.DBX  124.7;
      A     #RRel;
      =     DB260.DBX  988.0;

      AN    DB1815.DBX   28.5; // Caustic Full --> Drain
      A     DB260.DBX  748.0;
      R     DB260.DBX  748.0;
      S     DB260.DBX  988.0;

      AN    DB1825.DBX   28.5; // Acid Full --> Drain
      A     DB260.DBX  828.0;
      R     DB260.DBX  828.0;
      S     DB260.DBX  988.0;

      AN    DB1835.DBX   28.5; // HWater Full --> Drain
      A     DB260.DBX  908.0;
      R     DB260.DBX  908.0;
      S     DB260.DBX  988.0;


// Message Destination Not Ready
      A(    ;
      AN    DB1815.DBX   28.5;
      A     #S2I.SFM28.I01;
      )     ;
      O(    ;
      AN    DB1825.DBX   28.5;
      A     #S2I.SFM28.I02;
      )     ;
      O(    ;
      AN    DB1835.DBX   28.5;
      A     #S2I.SFM28.I03;
      )     ;
      O(    ;
      AN    DB1845.DBX   28.5;
      A     #S2I.SFM28.I04;
      )     ;
      A     DB165.DBX  125.0; // Run Release
      JCN   DNRM;
      SET   ;
      R     DB165.DBX   27.7; // Run Release
      L     903; // Destination Not Ready
      T     MD    90;
DNRM: NOP   0;

// ---------------------------------------------------------------------------
// CIP Prerun ---
// ---------------------------------------------------------------------------
      L     DB165.DBD  142;
      T     #U.Seq.SFM[27].Sp;

// Caustic
      A     DB1815.DBX   27.7;
      A     DB165.DBX  124.6;
      A     #S2I.SFM27.I02;
      A     #RRel;
      =     DB260.DBX  668.0;

// Acid
      A     DB1825.DBX   27.7;
      A     DB165.DBX  124.6;
      A     #S2I.SFM27.I04;
      A     #RRel;
      =     DB260.DBX  588.0;

// Hot Water
      A     DB1835.DBX   27.7;
      A     DB165.DBX  124.6;
      A     #S2I.SFM27.I13;
      A     #RRel;
      =     DB260.DBX  508.0;

// Fresh Water
      A     DB1845.DBX   27.7;
      A     DB165.DBX  124.6;
      A     #S2I.SFM27.I12;
      A     #RRel;
      =     DB260.DBX  428.0;

// Pump
      A     DB165.DBX  124.6;
      A     DB165.DBX  125.3;
      AN    #S2I.SFM27.I00;
      A     #RRel;
      =     DB260.DBX  108.0;

      A     DB260.DBX  103.4;
      A     M    102.3;
      =     DB165.DBX   28.3;

// Steam Valve
      A     DB263.DBX  138.6;
      R     #U.Seq.User.Bit16;

      A     DB263.DBX  138.5;
      S     #U.Seq.User.Bit16;

      L     #U.Seq.SFM[36].Sp;
      L     0.000000e+000;
      >R    ;
      AN    #S2I.SFM27.I12; // Fresh Water
      AN    #U.Seq.User.Bit16;
//      A     "C06ActD".RV_P1.VOn     // Probleme mit start / stop
      A     #RRel;
      =     DB260.DBX  348.0;

// Message Source Not Ready
      AN    DB1815.DBX   27.7;
      AN    DB1825.DBX   27.7;
      AN    DB1835.DBX   27.7;
      AN    DB1845.DBX   27.7;
      A     DB165.DBX  124.6;
      AN    #S2I.SFM27.I00;
      JCN   SNRM;
      SET   ;
      R     DB165.DBX   27.5;
      L     904; // Source Not Ready
      T     MD    90;
SNRM: NOP   0;

// ---------------------------------------------------------------------------
// CIP Way ---
// ---------------------------------------------------------------------------
      L     #U.Seq.SFM[25].Sp;
      T     DB165.DBD   30;

// ---------------------------------------------------------------------------
// transition condition
      A     DB165.DBX  125.7;
      =     M    102.1;

// subphase evaluation
      L     MW   110;
      JL    D100;
      JU    COMM; // subphase  0:
// ---------------------------------------------------------------------------
D100: SET   ;
      S     M    110.7; // Error unknown subphase
      JU    COMM;

NETWORK
TITLE =End Of Sequence Organisation

COMM: SET   ;

// ---------------------------------------------------------------------------
// pause timer unit parameter


NETWORK
TITLE =General Post Phase Controls

      NOP   0;

// ---------------------------------------------------------------------------
// general postphase controls

//Write Temperature CIP Prerun from Master CIP Unit
      L     DB165.DBD  134;
      T     #U.Seq.SFM[36].Sp;

NETWORK
TITLE =Process Status Management

      NOP   0;

// ---------------------------------------------------------------------------
// Signal Control
// -------------------------------------------------
// Maintenance
// -------------------------------------------------
// CIP Required
// -------------------------------------------------
// CIP Active
// -------------------------------------------------
// CIP Clean
// -------------------------------------------------
// SIP Required
// -------------------------------------------------
// SIP Active
// -------------------------------------------------
// SIP Clean
// -------------------------------------------------
// Full
// -------------------------------------------------
// Filling
// -------------------------------------------------
// Ready For Filling
// -------------------------------------------------
// Empty
// -------------------------------------------------
// Emptying
// -------------------------------------------------
// Ready For Emptying
// -------------------------------------------------
// Reserved
// -------------------------------------------------
// Production
// -------------------------------------------------
// Used
// -------------------------------------------------
// PStat Function Call
//      CALL  "PStat"
//       UnitNo     :=#UnitNo
//       PStatModVal:="C06UnVD".unv001.ValExt


NETWORK
TITLE =Unit Hold Request and Messages

      SET   ;

// ---------------------------------------------------------------------------
// Set unit to "hold" if maintenance
      AN    #U.Seq.Switch.Sw31; // maintenance !
      JC    NCO1;
      S     M    120.3;
      L     998; // "Unit in maintenance !"
      T     MD    90;

// ---------------------------------------------------------------------------
// Set unit to "hold" if emergency stop
NCO1: A     #EStopOK;
      JC    NCO2;
      S     M    120.3;
      L     999; // "Emergency stop !"
      T     MD    90;
NCO2: NOP   0;

END_FUNCTION_BLOCK

FUNCTION_BLOCK FB 163
TITLE =C06: CIP Line x
AUTHOR : Woermann
NAME : C06Rel
VERSION : 0.1


VAR
  U : UDT 111;
END_VAR
VAR_TEMP
  CIP : BOOL ;	//CIP active
  UNIM : BOOL ;	//Unit Not In Maintenance
  GenRel : BOOL ;	//general OK (emergency and maintenance OK)
  EStopOK : BOOL ;	//emergency OK
  UnitNo : INT ;	//unit number
  xTmp : BOOL ;	//Temporary Bool
  iTmp : INT ;	//Temporary INT
  rTmp : REAL ;	//Temporary REAL
  dTmp : DINT ;	//Temporary DINT (free for general use)
  RetValInt : INT ;	//return value
END_VAR
BEGIN
NETWORK
TITLE =General

      SET   ;
// Simulation ---------------------------------------------------------------
      A     #U.Seq.User.Bit63;
      CC    FB   169; // "C06Sim"
      A     #U.Seq.Sim;
      =     #U.Seq.User.Bit63; //Help bit for simulation

// get unit number ----------------------------------------------------------
      L     MB   112;
      T     #UnitNo;

// CIP ----------------------------------------------------------------------
      L     #U.Seq.ProgNo;
      L     0;
      <D    ;
      =     #CIP;

// emergency OK -------------------------------------------------------------
      A     DB165.DBX   27.0; //Emergency Stop OK
      =     #EStopOK;

// Write Unit in Maintenance ------------------------------------------------

      AN    #U.Seq.Switch.Sw31;
      =     #UNIM;

// emergency and maintenance OK ---------------------------------------------
      A     #EStopOK;
      A     #UNIM;
      =     #GenRel;

// communication ------------------------------------------------------------
      UC    FB   165; // U091Com

NETWORK
TITLE =Analog Inputs

      NOP   0;

// ----------------------------------------------------------
// RV1T1 Regler 2 RV 1 Temperatur 1
// ----------------------------------------------------------
      L     #U.Seq.SFM[63].Sp; // !!! insert correct SFM !!!
      T     DB263.DBD  238;

      SET   ;
      =     DB263.DBX  141.5;

// ----------------------------------------------------------
// TI_RR1 Temperatur CIP Rücklauf 1
// ----------------------------------------------------------
      L     #U.Seq.SFM[63].Sp; // !!! insert correct SFM !!!
      T     DB263.DBD  358;

      SET   ;
      =     DB263.DBX  261.5;

// ----------------------------------------------------------
// CS_RR1 Messbereich ist umschaltber
// ----------------------------------------------------------
      L     #U.Seq.SFM[63].Sp; // !!! insert correct SFM !!!
      T     DB263.DBD  478;

      SET   ;
      =     DB263.DBX  381.5;

// ----------------------------------------------------------
// FIT_RV1 Flow CIP Kreislauf 1
// ----------------------------------------------------------
      L     #U.Seq.SFM[63].Sp; // !!! insert correct SFM !!!
      T     DB263.DBD  598;

      SET   ;
      =     DB263.DBX  501.5;

NETWORK
TITLE =Universal Value

      NOP   0;

// ----------------------------------------------------------
// unv001 Process Status
// ----------------------------------------------------------
// process value to UnV
//      L     0.000000e+000
//      T     "C06UnVD".unv001.ValExt

// ----------------------------------------------------------
// unv002 Universal Value 02
// ----------------------------------------------------------
// process value to UnV
//      L     0.000000e+000
//      T     "C06UnVD".unv002.ValExt

NETWORK
TITLE =Special Input

      NOP   0;

// ----------------------------------------------------------
// FS_RR1_NEU
// ----------------------------------------------------------
      AN    DB165.DBX   24.7;
      A     DB165.DBX   24.0;
      A     DB165.DBX  125.4;
      =     DB261.DBX   81.4;
      SET   ;
      =     DB261.DBX   81.5;

// ----------------------------------------------------------
// IDM_IMPULSE_RV_1FQS DURCHFLUSSMESSUNG KREISLAUF 1
// ----------------------------------------------------------
      CLR   ;
//      =     "C06SpID".IDM_IMPULSE_RV_1FQS.EAl
//      =     "C06SpID".IDM_IMPULSE_RV_1FQS.Pre

NETWORK
TITLE =Messages

      NOP   0;

// ----------------------------------------------------------
// msg001 Message 01
// ----------------------------------------------------------
      SET   ;
      R     DB267.DBX   80.7;
      =     DB267.DBX   81.4;

      CLR   ;
      =     DB267.DBX   82.7;

// ----------------------------------------------------------
// msg002 Message 02
// ----------------------------------------------------------
      SET   ;
      R     DB267.DBX  140.7;
      =     DB267.DBX  141.4;

      CLR   ;
      =     DB267.DBX  142.7;

NETWORK
TITLE =Counters
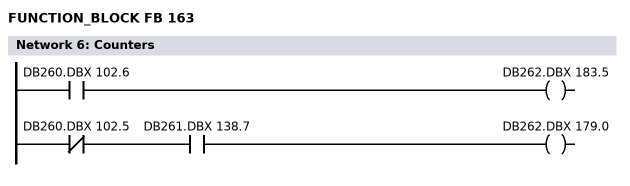

      NOP   0;

// ----------------------------------------------------------
// IDM_IMPULSE_RV_1FQI DURCHFLUSSMESSUNG KREISLAUF 1 (U91)
// ----------------------------------------------------------
      A     DB260.DBX  102.6;
      =     DB262.DBX  183.5;

      AN    DB260.DBX  102.5;
      A     DB261.DBX  138.7;
      =     DB262.DBX  179.0;

NETWORK
TITLE =PID controller

      NOP   0;

// ----------------------------------------------------------
// RV1RV CIP 1
// ----------------------------------------------------------
// starting value -----------------------
      A     DB260.DBX  343.4;
      A     #GenRel;
      =     DB266.DBX  203.2;
      =     DB266.DBX  203.5;

// enable alarm -------------------------
      A     DB266.DBX  203.5;
      A     DB266.DBX  201.4;
      AN    DB266.DBX  203.1;
      AN    DB266.DBX  203.3;
      AN    DB266.DBX  203.4;
      =     DB266.DBX  203.0;

// setpoint to controller ---------------
      L     #U.Seq.SFM[36].Sp; // CIP Prerun Temperature
      L     DB165.DBD  134;
      T     DB266.DBD  234;

// static value to controller ----------
      L     #U.Seq.SFM[63].Sp; // !!! insert correct SFM !!!
      T     DB266.DBD  238;

// process value to controller ----------
      L     DB263.DBD  146;
      T     DB266.DBD  254;

// low/high value to controller ---------
      L     DB263.DBD  150;
      T     DB266.DBD  218;

      L     DB263.DBD  154;
      T     DB266.DBD  222;

      L     DB263.DBD  506;
      T     DB266.DBD  310;
NETWORK
TITLE =Sequence organisation

// SFM supply ----------------------------------------------------------------

// analog value to SFM Regler 2 RV 1 Temperatur 1 -----------------------
      L     DB263.DBD  146;
      T     #U.Seq.SFM[36].Val; // CIP Prerun Temperature

// analog value to SFM Temperatur CIP Rücklauf 1 -----------------------
      L     DB263.DBD  266;
      T     #U.Seq.SFM[30].Val; // CIP Return Temperature

// analog value to SFM Messbereich ist umschaltber -----------------------
      L     DB263.DBD  386;
      T     #U.Seq.SFM[32].Val; // CIP Return Conductivity

// analog value to SFM Flow CIP Kreislauf 1 -----------------------
      L     DB263.DBD  506;
      T     #U.Seq.SFM[34].Val; // CIP Prerun Flow

NETWORK
TITLE =Auto / Manual

      SET   ;
      AN    M    122.2;
      JC    MODE;
      AN    M    120.1;

// assign actuator mode
      AN    M    120.1;
      =     DB260.DBX  105.4;
      =     DB260.DBX  345.4;
      =     DB260.DBX  425.4;
      =     DB260.DBX  505.4;
      =     DB260.DBX  585.4;
      =     DB260.DBX  665.4;
      =     DB260.DBX  745.4;
      =     DB260.DBX  825.4;
      =     DB260.DBX  905.4;
      =     DB260.DBX  985.4;
      =     DB260.DBX 2585.4;
      =     DB260.DBX 2665.4;
      =     DB260.DBX 2745.4;

// assign PID mode
      S     DB266.DBX  201.4;
      S     DB266.DBX  201.5;


MODE: SET   ;

NETWORK
TITLE =RV_P1 Reinigungsvorlaufpumpe Kreis 1
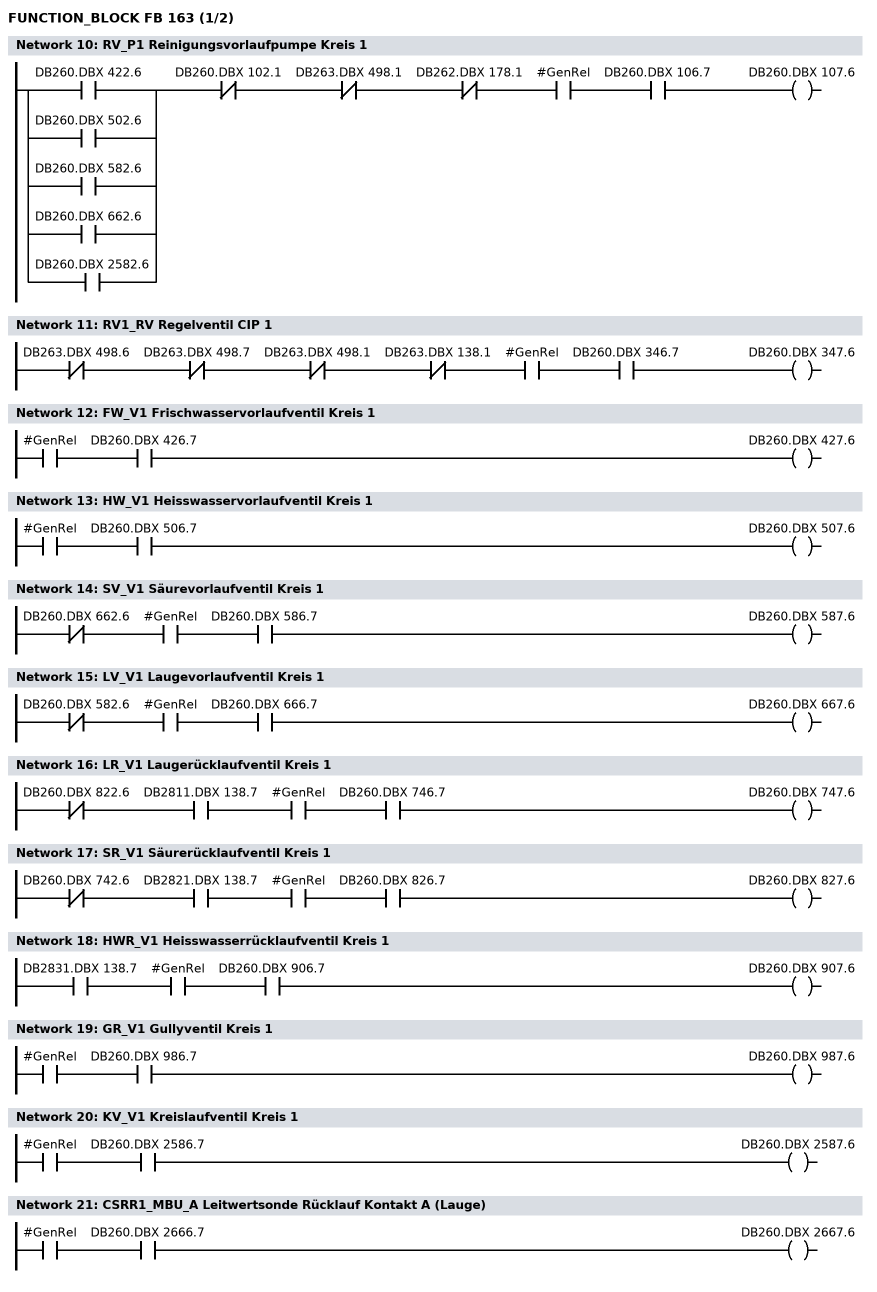

      O     DB260.DBX  422.6;
      O     DB260.DBX  502.6;
      O     DB260.DBX  582.6;
      O     DB260.DBX  662.6;
      O     DB260.DBX 2582.6;

      AN    DB260.DBX  102.1;
      AN    DB263.DBX  498.1;
      AN    DB262.DBX  178.1;

      A     #GenRel;
      A     DB260.DBX  106.7;
      =     DB260.DBX  107.6;
NETWORK
TITLE =RV1_RV Regelventil CIP 1

//      A     "C06ActD".RV_P1.VOn
      AN    DB263.DBX  498.6;
      AN    DB263.DBX  498.7;
      AN    DB263.DBX  498.1;
      AN    DB263.DBX  138.1;
      A     #GenRel;
      A     DB260.DBX  346.7;
      =     DB260.DBX  347.6;
NETWORK
TITLE =FW_V1 Frischwasservorlaufventil Kreis 1

      A     #GenRel;
      A     DB260.DBX  426.7;
      =     DB260.DBX  427.6;
NETWORK
TITLE =HW_V1 Heisswasservorlaufventil Kreis 1

      A     #GenRel;
      A     DB260.DBX  506.7;
      =     DB260.DBX  507.6;
NETWORK
TITLE =SV_V1 Säurevorlaufventil Kreis 1

      AN    DB260.DBX  662.6;

      A     #GenRel;
      A     DB260.DBX  586.7;
      =     DB260.DBX  587.6;
NETWORK
TITLE =LV_V1 Laugevorlaufventil Kreis 1

      AN    DB260.DBX  582.6;

      A     #GenRel;
      A     DB260.DBX  666.7;
      =     DB260.DBX  667.6;
NETWORK
TITLE =LR_V1 Laugerücklaufventil Kreis 1

      AN    DB260.DBX  822.6;

      A     DB2811.DBX  138.7;

      A     #GenRel;
      A     DB260.DBX  746.7;
      =     DB260.DBX  747.6;
NETWORK
TITLE =SR_V1 Säurerücklaufventil Kreis 1

      AN    DB260.DBX  742.6;

      A     DB2821.DBX  138.7;

      A     #GenRel;
      A     DB260.DBX  826.7;
      =     DB260.DBX  827.6;
NETWORK
TITLE =HWR_V1 Heisswasserrücklaufventil Kreis 1

      A     DB2831.DBX  138.7;

      A     #GenRel;
      A     DB260.DBX  906.7;
      =     DB260.DBX  907.6;
NETWORK
TITLE =GR_V1 Gullyventil Kreis 1

      A     #GenRel;
      A     DB260.DBX  986.7;
      =     DB260.DBX  987.6;
NETWORK
TITLE =KV_V1 Kreislaufventil Kreis 1

      A     #GenRel;
      A     DB260.DBX 2586.7;
      =     DB260.DBX 2587.6;
NETWORK
TITLE =CSRR1_MBU_A Leitwertsonde Rücklauf Kontakt A (Lauge)

      A     #GenRel;
      A     DB260.DBX 2666.7;
      =     DB260.DBX 2667.6;
NETWORK
TITLE =CSRR1_MBU_B Leitwertsonde Rücklauf Kontakt B (Saure)
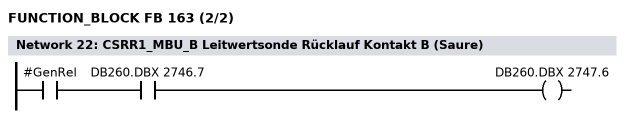

      A     #GenRel;
      A     DB260.DBX 2746.7;
      =     DB260.DBX 2747.6;
END_FUNCTION_BLOCK

FUNCTION_BLOCK FB 171
TITLE =C07: Brunnen Transfer Plan
// NW  1 : phase and index evaluation
// NW  2 : phase  1: Startposition
// NW  3 : phase 19: Plananpassung
// NW  4 : end of sequence
// NW  5 : unit hold request
//SFM   Use                                 Datatype        UoM
//----+-------------------------------------------------------------------------
// 09 : Prozesszeit                         Dauer           min
// 10 : Aktueller Tank                      Equipment
// 11 : 1. Tank                             Equipment
// 12 : 2. Tank                             Equipment
// 13 : 3. Tank                             Equipment
// 14 : Quelle                              Equipment
// 16 : Menge                               Wert            m3
// 22 : pH                                  Wert            pH
// 23 : Chriwa Status 1                     Aufzählung
// 24 : Chriwa Status 2                     Aufzählung
// 42 : Material                            Material
AUTHOR : Woermann
NAME : C06Seq
VERSION : 0.1
CODE_VERSION1


VAR
  U : UDT 161;
END_VAR
VAR_TEMP
  CIP : BOOL ;	//CIP active
  ComCIP : BOOL ;	//Communication With CIP Active
  ComDST : BOOL ;	//Communication With DST OK (Same Mat)
  RRel : BOOL ;	//Run Release
  EStopOK : BOOL ;	//emergency OK
  StepMax : BOOL ;	//StepMax (last) active
  SubStepMax : BOOL ;	//SubStepMax (last) active
  SubStepMaxD : BOOL ;	//SubStepMax (last) done
  ChkOK : BOOL ;	//SubStepMax (last) done
  xTmp : BOOL ;	//Temporary BOOL (free for general use)
  iTmp : INT ;	//Temporary INT (free for general use)
  dTmp : DINT ;	//Temporary DINT (free for general use)
  rTmp : REAL ;	//Temporary REAL (free for general use)
  UnitNo : INT ;	//Unit Number
  EquipmentID : INT ;	//Equipment ID
  S2I : STRUCT 	//SFM to indexes
   SFM10 : STRUCT 	//Aktueller Tank
    I00 : BOOL ;	//Bitte auswählen
    I01 : BOOL ;
    I02 : BOOL ;
    I03 : BOOL ;
    I04 : BOOL ;
    I05 : BOOL ;
    I06 : BOOL ;
    I07 : BOOL ;
    I08 : BOOL ;
    I09 : BOOL ;
    I10 : BOOL ;
    I11 : BOOL ;
    I12 : BOOL ;
    I13 : BOOL ;
    I14 : BOOL ;
    I15 : BOOL ;
    I16 : BOOL ;
    I17 : BOOL ;
    I18 : BOOL ;
    I19 : BOOL ;
    I20 : BOOL ;
    I21 : BOOL ;
    I22 : BOOL ;
    I23 : BOOL ;
    I24 : BOOL ;
    I25 : BOOL ;
    I26 : BOOL ;
    I27 : BOOL ;
    I28 : BOOL ;
    I29 : BOOL ;
    I30 : BOOL ;
    I31 : BOOL ;
   END_STRUCT ;
   SFM11 : STRUCT 	//1. Tank
    I00 : BOOL ;	//Bitte auswählen
    I01 : BOOL ;
    I02 : BOOL ;
    I03 : BOOL ;
    I04 : BOOL ;
    I05 : BOOL ;
    I06 : BOOL ;
    I07 : BOOL ;
    I08 : BOOL ;
    I09 : BOOL ;
    I10 : BOOL ;
    I11 : BOOL ;
    I12 : BOOL ;
    I13 : BOOL ;
    I14 : BOOL ;
    I15 : BOOL ;
    I16 : BOOL ;
    I17 : BOOL ;
    I18 : BOOL ;
    I19 : BOOL ;
    I20 : BOOL ;
    I21 : BOOL ;
    I22 : BOOL ;
    I23 : BOOL ;
    I24 : BOOL ;
    I25 : BOOL ;
    I26 : BOOL ;
    I27 : BOOL ;
    I28 : BOOL ;
    I29 : BOOL ;
    I30 : BOOL ;
    I31 : BOOL ;
   END_STRUCT ;
   SFM12 : STRUCT 	//2. Tank
    I00 : BOOL ;	//Bitte auswählen
    I01 : BOOL ;
    I02 : BOOL ;
    I03 : BOOL ;
    I04 : BOOL ;
    I05 : BOOL ;
    I06 : BOOL ;
    I07 : BOOL ;
    I08 : BOOL ;
    I09 : BOOL ;
    I10 : BOOL ;
    I11 : BOOL ;
    I12 : BOOL ;
    I13 : BOOL ;
    I14 : BOOL ;
    I15 : BOOL ;
    I16 : BOOL ;
    I17 : BOOL ;
    I18 : BOOL ;
    I19 : BOOL ;
    I20 : BOOL ;
    I21 : BOOL ;
    I22 : BOOL ;
    I23 : BOOL ;
    I24 : BOOL ;
    I25 : BOOL ;
    I26 : BOOL ;
    I27 : BOOL ;
    I28 : BOOL ;
    I29 : BOOL ;
    I30 : BOOL ;
    I31 : BOOL ;
   END_STRUCT ;
   SFM13 : STRUCT 	//3. Tank
    I00 : BOOL ;	//Bitte auswählen
    I01 : BOOL ;
    I02 : BOOL ;
    I03 : BOOL ;
    I04 : BOOL ;
    I05 : BOOL ;
    I06 : BOOL ;
    I07 : BOOL ;
    I08 : BOOL ;
    I09 : BOOL ;
    I10 : BOOL ;
    I11 : BOOL ;
    I12 : BOOL ;
    I13 : BOOL ;
    I14 : BOOL ;
    I15 : BOOL ;
    I16 : BOOL ;
    I17 : BOOL ;
    I18 : BOOL ;
    I19 : BOOL ;
    I20 : BOOL ;
    I21 : BOOL ;
    I22 : BOOL ;
    I23 : BOOL ;
    I24 : BOOL ;
    I25 : BOOL ;
    I26 : BOOL ;
    I27 : BOOL ;
    I28 : BOOL ;
    I29 : BOOL ;
    I30 : BOOL ;
    I31 : BOOL ;
   END_STRUCT ;
   SFM14 : STRUCT 	//Quelle
    I00 : BOOL ;	//Bitte auswählen
    I01 : BOOL ;
    I02 : BOOL ;
    I03 : BOOL ;
    I04 : BOOL ;
    I05 : BOOL ;
    I06 : BOOL ;
    I07 : BOOL ;
    I08 : BOOL ;
    I09 : BOOL ;
    I10 : BOOL ;
    I11 : BOOL ;
    I12 : BOOL ;
    I13 : BOOL ;
    I14 : BOOL ;
    I15 : BOOL ;
    I16 : BOOL ;
    I17 : BOOL ;
    I18 : BOOL ;
    I19 : BOOL ;
    I20 : BOOL ;
    I21 : BOOL ;
    I22 : BOOL ;
    I23 : BOOL ;
    I24 : BOOL ;
    I25 : BOOL ;
    I26 : BOOL ;
    I27 : BOOL ;
    I28 : BOOL ;
    I29 : BOOL ;
    I30 : BOOL ;
    I31 : BOOL ;
   END_STRUCT ;
   SFM23 : STRUCT 	//Chriwa Status 1
    I00 : BOOL ;	//Erstfiltrat
    I01 : BOOL ;	//Aus
    I02 : BOOL ;	//Bereitschaft
    I03 : BOOL ;	//Stop
    I04 : BOOL ;	//Störung
    I05 : BOOL ;
    I06 : BOOL ;
    I07 : BOOL ;
    I08 : BOOL ;	//Betrieb
    I09 : BOOL ;	//Entspannen
    I10 : BOOL ;	//Absenken
    I11 : BOOL ;	//Spülen Luft
    I12 : BOOL ;	//Spülen Wasser/Luft
    I13 : BOOL ;	//Filterbettentleerung
    I14 : BOOL ;	//Spülen Wasser
    I15 : BOOL ;	//Auffüllen
    I16 : BOOL ;	//Nicht definiert
    I17 : BOOL ;
    I18 : BOOL ;
    I19 : BOOL ;
    I20 : BOOL ;
    I21 : BOOL ;
    I22 : BOOL ;
    I23 : BOOL ;
    I24 : BOOL ;
    I25 : BOOL ;
    I26 : BOOL ;
    I27 : BOOL ;
    I28 : BOOL ;
    I29 : BOOL ;
    I30 : BOOL ;
    I31 : BOOL ;
   END_STRUCT ;
   SFM24 : STRUCT 	//Chriwa Status 2
    I00 : BOOL ;	//Erstfiltrat
    I01 : BOOL ;	//Aus
    I02 : BOOL ;	//Bereitschaft
    I03 : BOOL ;	//Stop
    I04 : BOOL ;	//Störung
    I05 : BOOL ;
    I06 : BOOL ;
    I07 : BOOL ;
    I08 : BOOL ;	//Betrieb
    I09 : BOOL ;	//Entspannen
    I10 : BOOL ;	//Absenken
    I11 : BOOL ;	//Spülen Luft
    I12 : BOOL ;	//Spülen Wasser/Luft
    I13 : BOOL ;	//Filterbettentleerung
    I14 : BOOL ;	//Spülen Wasser
    I15 : BOOL ;	//Auffüllen
    I16 : BOOL ;	//Nicht definiert
    I17 : BOOL ;
    I18 : BOOL ;
    I19 : BOOL ;
    I20 : BOOL ;
    I21 : BOOL ;
    I22 : BOOL ;
    I23 : BOOL ;
    I24 : BOOL ;
    I25 : BOOL ;
    I26 : BOOL ;
    I27 : BOOL ;
    I28 : BOOL ;
    I29 : BOOL ;
    I30 : BOOL ;
    I31 : BOOL ;
   END_STRUCT ;
   SFM39 : STRUCT 	//Q-Status
    I00 : BOOL ;	//Bitte auswählen
    I01 : BOOL ;	//freigegeben
    I02 : BOOL ;
    I03 : BOOL ;
    I04 : BOOL ;
    I05 : BOOL ;
    I06 : BOOL ;	//ignorieren
    I07 : BOOL ;
    I08 : BOOL ;
    I09 : BOOL ;	//gesperrt
    I10 : BOOL ;
    I11 : BOOL ;
    I12 : BOOL ;
    I13 : BOOL ;
    I14 : BOOL ;
    I15 : BOOL ;
    I16 : BOOL ;
    I17 : BOOL ;
    I18 : BOOL ;
    I19 : BOOL ;
    I20 : BOOL ;
    I21 : BOOL ;
    I22 : BOOL ;
    I23 : BOOL ;
    I24 : BOOL ;
    I25 : BOOL ;
    I26 : BOOL ;
    I27 : BOOL ;
    I28 : BOOL ;
    I29 : BOOL ;
    I30 : BOOL ;
    I31 : BOOL ;
   END_STRUCT ;
  END_STRUCT ;
END_VAR
BEGIN
NETWORK
TITLE = Phase and Index Evaluation

      CLR   ;
      =     #RRel;
      =     DB175.DBX   27.6;

      L     0;
      T     DB175.DBD   30;
      T     DB175.DBD   34;
      T     DB175.DBD   38;
      T     DB175.DBD   42;
      T     DB175.DBD   46;

// ---------------------------------------------------------------------------
// write max used SFM's (last SFM number + 1)
      L     43;
      T     #U.SFMQuant;

// ---------------------------------------------------------------------------
// unit & equipment number
      L     MB   112;
      T     #UnitNo;

      L     DB175.DBW   14;
      L     1000;
      *I    ;
      L     #UnitNo;
      +I    ;
      T     #EquipmentID;

// ---------------------------------------------------------------------------
// CIP active
      L     MW   114;
      L     0;
      <I    ;
      =     #CIP;

// ---------------------------------------------------------------------------
// communicating units
      CLR   ;
      =     #ComCIP;

// ---------------------------------------------------------------------------
// process timer start
      SET   ;
      =     M    131.0;

// ---------------------------------------------------------------------------
// emergency OK
      A     DB175.DBX   27.0;
      =     #EStopOK;

// define last (Sub)Step active
      L     #U.Seq.StepMax;
      L     MW   104;
      ==I   ;
      =     #StepMax;

      L     #U.Seq.SubStepMax;
      L     MW   118;
      ==I   ;
      =     #SubStepMax;

      A     #SubStepMax;
      A     #U.Seq.SPD;
      AN    M    103.2;
      =     #SubStepMaxD;


// ---------------------------------------------------------------------------
// phase evaluation
      L     MW   108;
      JL    X0;
      JU    X0; // phase  0:
      JU    X1; // phase  1: Startposition
      JU    X0; // phase  2:
      JU    X0; // phase  3: Vorspülen
      JU    X0; // phase  4: System befüllen
      JU    X0; // phase  5: Transfer
      JU    X0; // phase  6: Standby
      JU    X0; // phase  7:
      JU    X0; // phase  8: Ausschub
      JU    X0; // phase  9:
      JU    X0; // phase 10:
      JU    X0; // phase 11: Nachspülen
      JU    X0; // phase 12:
      JU    X0; // phase 13:
      JU    X0; // phase 14:
      JU    X0; // phase 15:
      JU    X0; // phase 16:
      JU    X0; // phase 17:
      JU    X0; // phase 18:
      JU    X19; // phase 19: Plananpassung
X0:   SET   ;
      S     M    108.7; // Error unknown phase
      JU    COMM;
NETWORK
TITLE =phase 1: startposition

X1:   SET   ;

// ---------------------------------------------------------------------------
// general functions
// ---------------------------------------------------------------------------
// reset signals
      A     M    102.2;
      R     #U.Seq.Switch.Sw1;
      R     #U.Seq.Switch.Sw2;

      AN    M    102.0;
      =     M    161.0; // Reset Process Timer

      CALL FC   709 (// Reset "Simulation" And "Ignore"
           UnitNo                   := #UnitNo,// Of All Control Modules
           Enable                   := M    102.2);// At First Cycle of Startposition (Idle)

// ---------------------------------------------------------------------------
// start check --------------------------------------------------------------
      A     #CIP;
      JC    M010;

      CALL FC   170 (
           ChkType                  := 1,// production
           ChkOK                    := M    122.0);
      JU    COMM;

M010: CALL FC   170 (
           ChkType                  := 2,// CIP
           ChkOK                    := M    122.0);
      JU    COMM;
NETWORK
TITLE =phase 19: Plananpassung
//SFM   Use                                 Datatype        UoM
//----+-------------------------------------------------------------------------
// 00 : Schrittüberwachzeit                 Dauer           min
// 16 : Menge                               Wert            kg
// 20 : Durchfluss                          Wert            m3/h
X19:  SET   ;
// ---------------------------------------------------------------------------
// General CM evaluation

// ---------------------------------------------------------------------------
// general functions
      AN    M    121.2;
      A     M    102.3;
      =     #RRel;

// ---------------------------------------------------------------------------
// messages
// ---------------------------------------------------------------------------
// timer & counter
      A     M    102.0;

// ---------------------------------------------------------------------------
// pause timer
// ---------------------------------------------------------------------------
// communication
      L     DB175.DBD  174;
      L     #U.Seq.SFM[42].Sp;
      ==R   ;
      AN    DB175.DBX  168.7;
      AN    DB175.DBX   24.7;
      =     #ComDST;

      A     #ComDST;
      A     M    102.3;
      S     DB175.DBX   29.0; // Request Data Copy
      AN    M    102.0;
      O     M    102.2;
      R     DB175.DBX   29.0; // Request Data Copy

      L     #U.Seq.SFM[42].Sp; // Mateial
      T     DB175.DBD   30;
      L     #U.Seq.SFM[16].Sp; // Menge
      T     DB175.DBD   34;
      L     #U.Seq.SFM[11].Sp; // Tank 1
      T     DB175.DBD   38;
      L     #U.Seq.SFM[12].Sp; // Tank 2
      T     DB175.DBD   42;
      L     #U.Seq.SFM[13].Sp; // Tank 3
      T     DB175.DBD   46;

// ---------------------------------------------------------------------------
// control modules
      A     M    102.3;

// ---------------------------------------------------------------------------
// transition condition
      L     #U.Seq.SFM[0].Val;
      L     1.000000e+000;
      >=R   ;
      A     #ComDST;
      A     DB175.DBX  173.0; // Data Copy Done
      =     M    102.1;

// subphase evaluation
      L     MW   110;
      JL    B900;
      JU    COMM; // subphase  0:
// ---------------------------------------------------------------------------
B900: SET   ;
      S     M    110.7; // Error unknown subphase
      JU    COMM;
NETWORK
TITLE =End Of Sequence Organisation

COMM: SET   ;

// ---------------------------------------------------------------------------
// pause timer unit parameter


NETWORK
TITLE =General Post Phase Controls

      NOP   0;

// ---------------------------------------------------------------------------
// general postphase controls


NETWORK
TITLE =Process Status Management
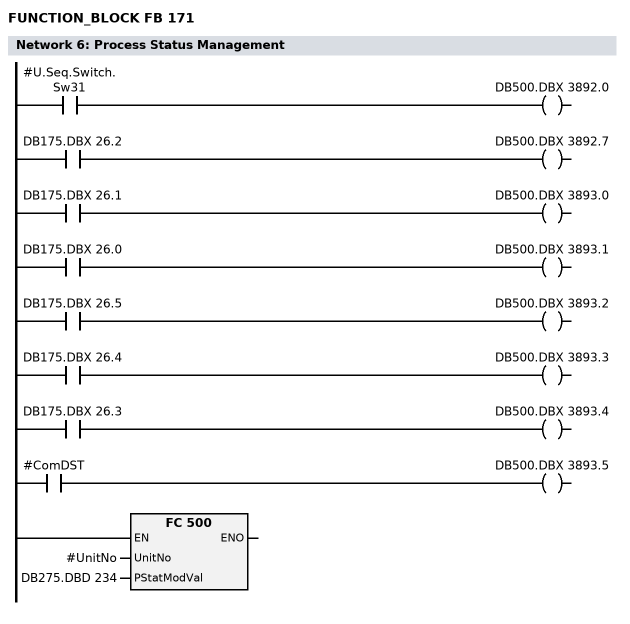

      NOP   0;
// ---------------------------------------------------------------------------
// Signal Control
// -------------------------------------------------
// Maintenance
      A     #U.Seq.Switch.Sw31;
      =     DB500.DBX 3892.0;
// -------------------------------------------------
// CIP Required
// -------------------------------------------------
// CIP Active
// -------------------------------------------------
// CIP Clean
// -------------------------------------------------
// SIP Required
// -------------------------------------------------
// SIP Active
// -------------------------------------------------
// SIP Clean
// -------------------------------------------------
// Full
      A     DB175.DBX   26.2;
      =     DB500.DBX 3892.7;
// -------------------------------------------------
// Filling
      A     DB175.DBX   26.1;
      =     DB500.DBX 3893.0;
// -------------------------------------------------
// Ready For Filling
      A     DB175.DBX   26.0;
      =     DB500.DBX 3893.1;
// -------------------------------------------------
// Empty
      A     DB175.DBX   26.5;
      =     DB500.DBX 3893.2;
// -------------------------------------------------
// Emptying
      A     DB175.DBX   26.4;
      =     DB500.DBX 3893.3;
// -------------------------------------------------
// Ready For Emptying
      A     DB175.DBX   26.3;
      =     DB500.DBX 3893.4;
// -------------------------------------------------
// Reserved
      A     #ComDST;
      =     DB500.DBX 3893.5;
// -------------------------------------------------
// Production
// -------------------------------------------------
// Used

// -------------------------------------------------
// PStat Function Call

      CALL FC   500 (
           UnitNo                   := #UnitNo,
           PStatModVal              := DB275.DBD  234);


NETWORK
TITLE =Unit Hold Request and Messages

      SET   ;

// ---------------------------------------------------------------------------
// Set unit to "hold" if maintenance
      AN    #U.Seq.Switch.Sw31; // maintenance !
      JC    NCO1;
      S     M    120.3;
      L     998; // "Unit in maintenance !"
      T     MD    90;

// ---------------------------------------------------------------------------
// Set unit to "hold" if emergency stop
NCO1: A     #EStopOK;
      JC    NCO2;
      S     M    120.3;
      L     999; // "Emergency stop !"
      T     MD    90;
NCO2: NOP   0;

END_FUNCTION_BLOCK

FUNCTION_BLOCK FB 173
TITLE =C07: Brunnen Transfer Plan
FAMILY : BOTEC_F1
NAME : U121E
VERSION : 1.2


VAR_TEMP
  CIP : BOOL ;	//CIP active
  UNIM : BOOL ;	//Unit Not In Maintenance
  GenRel : BOOL ;	//general OK (emergency and maintenance OK)
  EStopOK : BOOL ;	//emergency OK
  UnitNo : INT ;	//unit number
  xTmp : BOOL ;	//Temporary Bool
  iTmp : INT ;	//Temporary INT
  rTmp : REAL ;	//Temporary REAL
  dTmp : DINT ;	//Temporary DINT (free for general use)
  RetValInt : INT ;	//return value
END_VAR
BEGIN
NETWORK
TITLE =General

      SET   ;
// get unit number ----------------------------------------------------------
      L     DB170.DBW    0;
      T     #UnitNo;

// CIP ----------------------------------------------------------------------
      L     DB171.DBD   54;
      L     0;
      <D    ;
      =     #CIP;

// emergency OK -------------------------------------------------------------
      A     DB175.DBX   27.0; //Emergency Stop OK
      =     #EStopOK;

// Write Unit in Maintenance ------------------------------------------------

      AN    DB171.DBX   69.7;
      =     #UNIM;

// emergency and maintenance OK ---------------------------------------------
      A     #EStopOK;
      A     #UNIM;
      =     #GenRel;

// communication ------------------------------------------------------------
      UC    FB   175; // C07Com

NETWORK
TITLE =Analog Inputs

      NOP   0;

// ----------------------------------------------------------
// C_AnI01 spare
// ----------------------------------------------------------
      L     DB171.DBD 1118; // !!! insert correct SFM !!!
      T     DB273.DBD  238;

      CLR   ;
      =     DB273.DBX  141.5;
      =     DB273.DBX  140.6;
      =     DB273.DBX  140.7;

// ----------------------------------------------------------
// C_AnI002 spare
// ----------------------------------------------------------
      L     DB171.DBD 1118; // !!! insert correct SFM !!!
      T     DB273.DBD  358;

      CLR   ;
      =     DB273.DBX  261.5;
      =     DB273.DBX  260.6;
      =     DB273.DBX  260.7;

// ----------------------------------------------------------
// AnI03 spare
// ----------------------------------------------------------
      L     DB171.DBD 1118; // !!! insert correct SFM !!!
      T     DB273.DBD  478;

      CLR   ;
      =     DB273.DBX  381.5;
      =     DB273.DBX  380.6;
      =     DB273.DBX  380.7;

NETWORK
TITLE =Universal Value

      NOP   0;

// ----------------------------------------------------------
// unv001 Process Status
// ----------------------------------------------------------
// process value to UnV
//      L     0.000000e+000
//      T     "C07UnVD".unv001.ValExt

// ----------------------------------------------------------
// unv002 Universal Value 02
// ----------------------------------------------------------
// process value to UnV
//      L     0.000000e+000
//      T     "C07UnVD".unv002.ValExt

// ----------------------------------------------------------
// unv003 Druck Sollwert
// ----------------------------------------------------------
// process value to UnV
//      L     0.000000e+000
//      T     "C07UnVD".unv003.ValExt

// ----------------------------------------------------------
// unv004 Universal Value 04
// ----------------------------------------------------------
// process value to UnV
//      L     0.000000e+000
//      T     "C07UnVD".unv004.ValExt

NETWORK
TITLE =Special Input

      NOP   0;

// ----------------------------------------------------------
// SpI01 spare
// ----------------------------------------------------------
      SET   ;
      =     DB271.DBX   81.4;
      =     DB271.DBX   81.5;

// ----------------------------------------------------------
// SpI02 spare
// ----------------------------------------------------------
      SET   ;
      =     DB271.DBX  141.4;
      =     DB271.DBX  141.5;

// ----------------------------------------------------------
// SpI03 spare
// ----------------------------------------------------------
      SET   ;
      =     DB271.DBX  201.4;
      =     DB271.DBX  201.5;

// ----------------------------------------------------------
// SpI04 spare
// ----------------------------------------------------------
      SET   ;
      =     DB271.DBX  261.4;
      =     DB271.DBX  261.5;

NETWORK
TITLE =Messages

      NOP   0;

// ----------------------------------------------------------
// msg001 Message 01
// ----------------------------------------------------------
      SET   ;
      R     DB277.DBX   80.7;
      =     DB277.DBX   81.4;

      CLR   ;
      =     DB277.DBX   82.7;

// ----------------------------------------------------------
// msg002 Message 02
// ----------------------------------------------------------
      SET   ;
      R     DB277.DBX  140.7;
      =     DB277.DBX  141.4;

      CLR   ;
      =     DB277.DBX  142.7;

// ----------------------------------------------------------
// msg003 Message 03
// ----------------------------------------------------------
      SET   ;
      R     DB277.DBX  200.7;
      =     DB277.DBX  201.4;

      CLR   ;
      =     DB277.DBX  202.7;

NETWORK
TITLE =PID controller

      NOP   0;

// ----------------------------------------------------------
// PID01 spare
// ----------------------------------------------------------
// starting value -----------------------
//A     "C07ActD".Act.OutI // !!! insert correct Act !!!
      A     #GenRel;
      CLR   ;
      =     DB276.DBX  203.2;
      =     DB276.DBX  203.5;

// enable alarm -------------------------
      A     DB276.DBX  203.5;
      A     DB276.DBX  201.4;
      AN    DB276.DBX  203.1;
      AN    DB276.DBX  203.3;
      AN    DB276.DBX  203.4;
      =     DB276.DBX  203.0;

// setpoint to controller ---------------
      L     DB171.DBD 1118; // !!! insert correct SFM !!!
      T     DB276.DBD  234;

// static value to controller ----------
      L     DB171.DBD 1118; // !!! insert correct SFM !!!
      T     DB276.DBD  238;

// process value to controller ----------
      L     DB273.DBD   26; // !!! insert correct AnI !!!
      T     DB276.DBD  254;

